  Call Extruder(568.39008)
  MoveL 7921 to (479.59, 455.55, 140) mm, rotated rx -180 ry 0 rz 160 deg; joints [0.602, 52.757, 6.65, -156.409, 61.55, 168.248]
  Set speed (16.6 mm/s)
  Call Extruder(574.71594)
  MoveL 7922 to (481.3, 454.8, 140) mm, rotated rx 180 ry 0 rz 160 deg; joints [0.5, 53.008, 6.147, -156.467, 61.298, 168.187]
  Set speed (16.6 mm/s)
  Call Extruder(580.66586)
  MoveL 7923 to (482.93, 454.17, 140) mm, rotated rx 180 ry 0 rz 160 deg; joints [0.414, 53.249, 5.663, -156.511, 61.059, 168.124]
  Set speed (16.6 mm/s)
  Call Extruder(586.68166)
  MoveL 7924 to (484.6, 453.58, 140) mm, rotated rx -180 ry 0 rz 160 deg; joints [0.335, 53.498, 5.165, -156.544, 60.813, 168.053]
  Set speed (16.6 mm/s)
  Call Extruder(592.98031)
  MoveL 7925 to (486.37, 453.02, 140) mm, rotated rx 180 ry 0 rz 160 deg; joints [0.261, 53.764, 4.634, -156.568, 60.554, 167.972]
  Call Extruder(599.08597)
  MoveL 7926 to (488.1, 452.56, 140) mm, rotated rx -180 ry 0 rz 160 deg; joints [0.198, 54.026, 4.11, -156.579, 60.301, 167.887]
  Set speed (16.6 mm/s)
  Call Extruder(605.30009)
  MoveL 7927 to (489.88, 452.15, 140) mm, rotated rx -180 ry 0 rz 160 deg; joints [0.144, 54.297, 3.568, -156.579, 60.042, 167.794]
  Set speed (16.6 mm/s)
  Call Extruder(611.23622)
  MoveL 7928 to (491.6, 451.81, 140) mm, rotated rx -180 ry 0 rz 160 deg; joints [0.1, 54.56, 3.044, -156.568, 59.792, 167.699]
  Set speed (16.6 mm/s)
  Call Extruder(617.09230)
  MoveL 7929 to (493.3, 451.55, 140) mm, rotated rx -180 ry 0 rz 160 deg; joints [0.065, 54.822, 2.521, -156.547, 59.545, 167.598]
  Call Extruder(623.59424)
  MoveL 7930 to (495.2, 451.32, 140) mm, rotated rx 180 ry 0 rz 160 deg; joints [0.036, 55.117, 1.933, -156.511, 59.27, 167.479]
  Set speed (16.6 mm/s)
  Call Extruder(629.59472)
  MoveL 7931 to (496.97, 451.18, 140) mm, rotated rx -180 ry 0 rz 160 deg; joints [0.018, 55.391, 1.386, -156.466, 59.016, 167.363]
  Set speed (16.6 mm/s)
  Call Extruder(635.88670)
  MoveL 7932 to (498.82, 451.1, 140) mm, rotated rx 180 ry 0 rz 160 deg; joints [0.008, 55.682, 0.807, -156.409, 58.75, 167.235]
  Call Extruder(641.91456)
  MoveL 7933 to (500.59, 451.09, 140) mm, rotated rx -180 ry 0 rz 160 deg; joints [0.006, 55.963, 0.248, -156.343, 58.495, 167.105]
  Set speed (16.6 mm/s)
  Call Extruder(648.10941)
  MoveL 7934 to (502.41, 451.15, 140) mm, rotated rx 180 ry 0 rz 160 deg; joints [0.013, 56.253, -0.329, -156.263, 58.234, 166.966]
  Set speed (16.6 mm/s)
  Call Extruder(654.14645)
  MoveL 7935 to (504.19, 451.27, 140) mm, rotated rx 180 ry 0 rz 160 deg; joints [0.028, 56.538, -0.895, -156.175, 57.98, 166.823]
  Set speed (16.6 mm/s)
  Call Extruder(660.34108)
  MoveL 7936 to (506, 451.46, 140) mm, rotated rx 180 ry 0 rz 160 deg; joints [0.052, 56.831, -1.477, -156.074, 57.721, 166.67]
  Set speed (16.6 mm/s)
  Call Extruder(666.29236)
  MoveL 7937 to (507.73, 451.71, 140) mm, rotated rx 180 ry 0 rz 160 deg; joints [0.083, 57.113, -2.037, -155.967, 57.474, 166.517]
  Call Extruder(672.33230)
  MoveL 7938 to (509.48, 452.02, 140) mm, rotated rx -180 ry 0 rz 160 deg; joints [0.122, 57.4, -2.606, -155.849, 57.226, 166.356]
  Set speed (16.6 mm/s)
  Call Extruder(678.01374)
  MoveL 7939 to (511.12, 452.37, 140) mm, rotated rx -180 ry 0 rz 160 deg; joints [0.165, 57.669, -3.141, -155.729, 56.994, 166.2]
  Set speed (16.6 mm/s)
  Call Extruder(684.72563)
  MoveL 7940 to (513.03, 452.85, 140) mm, rotated rx 180 ry 0 rz 160 deg; joints [0.224, 57.988, -3.772, -155.575, 56.724, 166.008]
  Set speed (16.6 mm/s)
  Call Extruder(690.75124)
  MoveL 7941 to (514.73, 453.36, 140) mm, rotated rx -180 ry 0 rz 160 deg; joints [0.286, 58.273, -4.336, -155.427, 56.484, 165.83]
  Set speed (16.6 mm/s)
  Call Extruder(697.05633)
  MoveL 7942 to (516.49, 453.95, 140) mm, rotated rx 180 ry 0 rz 160 deg; joints [0.358, 58.57, -4.925, -155.263, 56.237, 165.638]
  Set speed (16.6 mm/s)
  Call Extruder(702.95462)
  MoveL 7943 to (518.12, 454.57, 140) mm, rotated rx 180 ry 0 rz 160 deg; joints [0.432, 58.847, -5.472, -155.1, 56.01, 165.453]
  Set speed (16.6 mm/s)
  Call Extruder(709.29068)
  MoveL 7944 to (519.84, 455.29, 140) mm, rotated rx -180 ry 0 rz 160 deg; joints [0.519, 59.143, -6.057, -154.916, 55.77, 165.248]
  Set speed (16.6 mm/s)
  Call Extruder(715.36245)
  MoveL 7945 to (521.45, 456.04, 140) mm, rotated rx 180 ry 0 rz 160 deg; joints [0.609, 59.424, -6.612, -154.731, 55.545, 165.048]
  Set speed (16.6 mm/s)
  Call Extruder(721.45875)
  MoveL 7946 to (523.05, 456.86, 140) mm, rotated rx -180 ry 0 rz 160 deg; joints [0.706, 59.703, -7.163, -154.537, 55.324, 164.842]
  Set speed (16.6 mm/s)
  Call Extruder(727.63337)
  MoveL 7947 to (524.64, 457.75, 140) mm, rotated rx -180 ry 0 rz 160 deg; joints [0.81, 59.983, -7.716, -154.332, 55.106, 164.628]
  Set speed (16.6 mm/s)
  Call Extruder(733.66477)
  MoveL 7948 to (526.16, 458.67, 140) mm, rotated rx 180 ry 0 rz 160 deg; joints [0.919, 60.253, -8.249, -154.124, 54.898, 164.415]
  Set speed (16.6 mm/s)
  Call Extruder(739.87872)
  MoveL 7949 to (527.68, 459.68, 140) mm, rotated rx 180 ry 0 rz 160 deg; joints [1.037, 60.528, -8.791, -153.903, 54.69, 164.192]
  Set speed (16.6 mm/s)
  Call Extruder(745.90071)
  MoveL 7950 to (529.13, 460.7, 140) mm, rotated rx -180 ry 0 rz 160 deg; joints [1.157, 60.79, -9.307, -153.681, 54.495, 163.972]
  Call Extruder(751.89968)
  MoveL 7951 to (530.53, 461.78, 140) mm, rotated rx 180 ry 0 rz 160 deg; joints [1.282, 61.046, -9.812, -153.454, 54.307, 163.75]
  Set speed (16.6 mm/s)
  Call Extruder(758.13508)
  MoveL 7952 to (531.94, 462.95, 140) mm, rotated rx 180 ry 0 rz 160 deg; joints [1.418, 61.308, -10.327, -153.212, 54.119, 163.516]
  Set speed (16.6 mm/s)
  Call Extruder(764.34204)
  MoveL 7953 to (533.3, 464.17, 140) mm, rotated rx -180 ry 0 rz 160 deg; joints [1.559, 61.562, -10.829, -152.964, 53.939, 163.28]
  Set speed (16.6 mm/s)
  Call Extruder(770.41574)
  MoveL 7954 to (534.59, 465.41, 140) mm, rotated rx -180 ry 0 rz 160 deg; joints [1.701, 61.806, -11.308, -152.716, 53.771, 163.047]
  Set speed (16.6 mm/s)
  Call Extruder(773.76102)
  MoveL 7955 to (535.27, 466.12, 140) mm, rotated rx 180 ry 0 rz 160 deg; joints [1.782, 61.937, -11.566, -152.578, 53.681, 162.918]
  Set speed (16.6 mm/s)
  Call Extruder(776.78327)
  MoveL 7956 to (535.89, 466.76, 140) mm, rotated rx 180 ry 0 rz 160 deg; joints [1.856, 62.055, -11.797, -152.452, 53.602, 162.801]
  Set speed (16.6 mm/s)
  Call Extruder(780.49101)
  MoveL 7957 to (536.62, 467.57, 140) mm, rotated rx 180 ry 0 rz 160 deg; joints [1.948, 62.197, -12.076, -152.295, 53.509, 162.657]
  Set speed (16.6 mm/s)
  Call Extruder(783.96552)
  MoveL 7958 to (537.29, 468.35, 140) mm, rotated rx -180 ry 0 rz 160 deg; joints [2.037, 62.327, -12.332, -152.147, 53.424, 162.522]
  Set speed (16.6 mm/s)
  Call Extruder(786.90697)
  MoveL 7959 to (537.84, 469.01, 140) mm, rotated rx -180 ry 0 rz 160 deg; joints [2.112, 62.436, -12.546, -152.02, 53.354, 162.407]
  Set speed (16.6 mm/s)
  Call Extruder(790.76461)
  MoveL 7960 to (538.55, 469.9, 140) mm, rotated rx 180 ry 0 rz 160 deg; joints [2.213, 62.576, -12.821, -151.853, 53.265, 162.256]
  Call Extruder(794.10006)
  MoveL 7961 to (539.15, 470.68, 140) mm, rotated rx 180 ry 0 rz 160 deg; joints [2.302, 62.694, -13.053, -151.707, 53.192, 162.125]
  Set speed (16.6 mm/s)
  Call Extruder(797.30570)
  MoveL 7962 to (539.71, 471.44, 140) mm, rotated rx 180 ry 0 rz 160 deg; joints [2.388, 62.806, -13.273, -151.566, 53.123, 162]
  Set speed (16.6 mm/s)
  Call Extruder(800.87078)
  MoveL 7963 to (540.31, 472.3, 140) mm, rotated rx 180 ry 0 rz 160 deg; joints [2.486, 62.928, -13.513, -151.408, 53.05, 161.86]
  Set speed (16.6 mm/s)
  Call Extruder(804.35419)
  MoveL 7964 to (540.88, 473.15, 140) mm, rotated rx -180 ry 0 rz 160 deg; joints [2.582, 63.045, -13.742, -151.253, 52.982, 161.724]
  Set speed (16.6 mm/s)
  Call Extruder(807.31812)
  MoveL 7965 to (541.35, 473.88, 140) mm, rotated rx 180 ry 0 rz 160 deg; joints [2.665, 63.142, -13.932, -151.121, 52.926, 161.608]
  Call Extruder(811.18100)
  MoveL 7966 to (541.95, 474.85, 140) mm, rotated rx -180 ry 0 rz 160 deg; joints [2.774, 63.265, -14.174, -150.947, 52.857, 161.457]
  Set speed (16.6 mm/s)
  Call Extruder(816.88134)
  MoveL 7967 to (542.79, 476.3, 140) mm, rotated rx -180 ry 0 rz 160 deg; joints [2.938, 63.441, -14.519, -150.69, 52.762, 161.236]
  Set speed (16.6 mm/s)
  Call Extruder(821.30516)
  MoveL 7968 to (543.4, 477.44, 140) mm, rotated rx 180 ry 0 rz 160 deg; joints [3.067, 63.572, -14.776, -150.489, 52.694, 161.065]
  Set speed (16.6 mm/s)
  Call Extruder(824.85035)
  MoveL 7969 to (543.87, 478.38, 140) mm, rotated rx -180 ry 0 rz 160 deg; joints [3.172, 63.674, -14.976, -150.327, 52.643, 160.929]
  Set speed (16.6 mm/s)
  Call Extruder(829.78773)
  MoveL 7970 to (544.5, 479.69, 140) mm, rotated rx 180 ry 0 rz 160 deg; joints [3.32, 63.81, -15.243, -150.102, 52.578, 160.74]
  Set speed (16.6 mm/s)
  Call Extruder(831.57607)
  MoveL 7971 to (544.71, 480.17, 140) mm, rotated rx 180 ry 0 rz 160 deg; joints [3.374, 63.858, -15.336, -150.02, 52.556, 160.673]
  Set speed (16.6 mm/s)
  Call Extruder(838.17107)
  MoveL 7972 to (545.46, 481.95, 140) mm, rotated rx -180 ry 0 rz 160 deg; joints [3.575, 64.027, -15.667, -149.719, 52.483, 160.424]
  Set speed (16.6 mm/s)
  Call Extruder(843.12930)
  MoveL 7973 to (545.98, 483.32, 140) mm, rotated rx 180 ry 0 rz 160 deg; joints [3.728, 64.146, -15.901, -149.492, 52.436, 160.241]
  Set speed (16.6 mm/s)
  Call Extruder(845.31622)
  MoveL 7974 to (546.19, 483.92, 140) mm, rotated rx 180 ry 0 rz 160 deg; joints [3.797, 64.196, -15.999, -149.393, 52.417, 160.16]
  Set speed (16.6 mm/s)
  Call Extruder(851.93089)
  MoveL 7975 to (546.8, 485.77, 140) mm, rotated rx 180 ry 0 rz 160 deg; joints [4.005, 64.341, -16.283, -149.091, 52.369, 159.92]
  Set speed (16.6 mm/s)
  Call Extruder(855.40941)
  MoveL 7976 to (547.08, 486.76, 140) mm, rotated rx -180 ry 0 rz 160 deg; joints [4.115, 64.411, -16.421, -148.933, 52.349, 159.796]
  Set speed (16.6 mm/s)
  Call Extruder(858.85943)
  MoveL 7977 to (547.35, 487.73, 140) mm, rotated rx 180 ry 0 rz 160 deg; joints [4.225, 64.479, -16.553, -148.777, 52.332, 159.674]
  Set speed (16.6 mm/s)
  Call Extruder(865.59259)
  MoveL 7978 to (547.81, 489.66, 140) mm, rotated rx -180 ry 0 rz 160 deg; joints [4.442, 64.6, -16.791, -148.473, 52.308, 159.44]
  Set speed (16.6 mm/s)
  Call Extruder(872.38173)
  MoveL 7979 to (548.19, 491.62, 140) mm, rotated rx -180 ry 0 rz 160 deg; joints [4.664, 64.708, -17.002, -148.17, 52.299, 159.212]
  Set speed (16.6 mm/s)
  Call Extruder(879.18152)
  MoveL 7980 to (548.49, 493.6, 140) mm, rotated rx 180 ry 0 rz 160 deg; joints [4.887, 64.802, -17.187, -147.869, 52.302, 158.99]
  Set speed (16.6 mm/s)
  Call Extruder(886.08891)
  MoveL 7981 to (548.72, 495.62, 140) mm, rotated rx -180 ry 0 rz 160 deg; joints [5.115, 64.883, -17.344, -147.568, 52.319, 158.774]
  Call Extruder(892.76703)
  MoveL 7982 to (548.85, 497.58, 140) mm, rotated rx 180 ry 0 rz 160 deg; joints [5.338, 64.947, -17.47, -147.281, 52.348, 158.572]
  Set speed (16.6 mm/s)
  Call Extruder(899.57193)
  MoveL 7983 to (548.91, 499.59, 140) mm, rotated rx 180 ry 0 rz 160 deg; joints [5.565, 64.998, -17.568, -146.993, 52.391, 158.376]
  Set speed (16.6 mm/s)
  Call Extruder(906.22719)
  MoveL 7984 to (548.89, 501.55, 140) mm, rotated rx 180 ry 0 rz 160 deg; joints [5.789, 65.032, -17.636, -146.717, 52.446, 158.193]
  Set speed (16.6 mm/s)
  Call Extruder(913.15085)
  MoveL 7985 to (548.78, 503.58, 140) mm, rotated rx -180 ry 0 rz 160 deg; joints [6.022, 65.053, -17.677, -146.436, 52.516, 158.013]
  Set speed (16.6 mm/s)
  Call Extruder(919.94097)
  MoveL 7986 to (548.59, 505.57, 140) mm, rotated rx 180 ry 0 rz 160 deg; joints [6.251, 65.059, -17.688, -146.167, 52.598, 157.847]
  Set speed (16.6 mm/s)
  Call Extruder(926.85256)
  MoveL 7987 to (548.32, 507.59, 140) mm, rotated rx -180 ry 0 rz 160 deg; joints [6.483, 65.049, -17.669, -145.9, 52.694, 157.689]
  Set speed (16.6 mm/s)
  Call Extruder(933.53369)
  MoveL 7988 to (547.98, 509.53, 140) mm, rotated rx 180 ry 0 rz 160 deg; joints [6.708, 65.025, -17.622, -145.648, 52.798, 157.547]
  Set speed (16.6 mm/s)
  Call Extruder(940.45609)
  MoveL 7989 to (547.54, 511.52, 140) mm, rotated rx -180 ry 0 rz 160 deg; joints [6.94, 64.984, -17.542, -145.396, 52.919, 157.413]
  Set speed (16.6 mm/s)
  Call Extruder(947.08762)
  MoveL 7990 to (547.04, 513.41, 140) mm, rotated rx 180 ry 0 rz 160 deg; joints [7.162, 64.931, -17.438, -145.162, 53.046, 157.295]
  Set speed (16.6 mm/s)
  Call Extruder(949.76693)
  MoveL 7991 to (546.82, 514.16, 140) mm, rotated rx 180 ry 0 rz 160 deg; joints [7.251, 64.905, -17.387, -145.07, 53.101, 157.251]
  Set speed (16.6 mm/s)
  Call Extruder(953.95077)
  MoveL 7992 to (546.45, 515.34, 140) mm, rotated rx 180 ry 0 rz 160 deg; joints [7.39, 64.861, -17.301, -144.928, 53.189, 157.185]
  Set speed (16.6 mm/s)
  Call Extruder(960.63540)
  MoveL 7993 to (545.79, 517.19, 140) mm, rotated rx -180 ry 0 rz 160 deg; joints [7.61, 64.778, -17.139, -144.709, 53.34, 157.091]
  Set speed (16.6 mm/s)
  Call Extruder(964.14755)
  MoveL 7994 to (545.42, 518.15, 140) mm, rotated rx 180 ry 0 rz 160 deg; joints [7.725, 64.729, -17.043, -144.597, 53.423, 157.046]
  Set speed (16.6 mm/s)
  Call Extruder(967.44744)
  MoveL 7995 to (545.05, 519.05, 140) mm, rotated rx 180 ry 0 rz 160 deg; joints [7.833, 64.681, -16.948, -144.493, 53.503, 157.005]
  Set speed (16.6 mm/s)
  Call Extruder(974.29011)
  MoveL 7996 to (544.23, 520.89, 140) mm, rotated rx -180 ry 0 rz 160 deg; joints [8.056, 64.568, -16.727, -144.285, 53.678, 156.932]
  Set speed (16.6 mm/s)
  Call Extruder(977.80399)
  MoveL 7997 to (543.77, 521.82, 140) mm, rotated rx 180 ry 0 rz 160 deg; joints [8.169, 64.504, -16.603, -144.182, 53.772, 156.9]
  Set speed (16.6 mm/s)
  Call Extruder(981.05322)
  MoveL 7998 to (543.34, 522.68, 140) mm, rotated rx 180 ry 0 rz 160 deg; joints [8.273, 64.443, -16.482, -144.088, 53.861, 156.873]
  Set speed (16.6 mm/s)
  Call Extruder(984.45482)
  MoveL 7999 to (542.87, 523.56, 140) mm, rotated rx -180 ry 0 rz 160 deg; joints [8.382, 64.374, -16.349, -143.993, 53.956, 156.848]
  Set speed (16.6 mm/s)
  Call Extruder(987.85938)
  MoveL 8000 to (542.38, 524.43, 140) mm, rotated rx 180 ry 0 rz 160 deg; joints [8.49, 64.303, -16.209, -143.899, 54.054, 156.825]
  Set speed (16.6 mm/s)
  Call Extruder(992.09448)
  MoveL 8001 to (541.74, 525.5, 140) mm, rotated rx -180 ry 0 rz 160 deg; joints [8.623, 64.21, -16.027, -143.786, 54.178, 156.802]
  Set speed (16.6 mm/s)
  Call Extruder(997.75133)
  MoveL 8002 to (540.85, 526.91, 140) mm, rotated rx -180 ry 0 rz 160 deg; joints [8.799, 64.077, -15.767, -143.642, 54.35, 156.778]
  Set speed (16.6 mm/s)
  Call Extruder(1002.84044)
  MoveL 8003 to (540, 528.15, 140) mm, rotated rx 180 ry 0 rz 160 deg; joints [8.955, 63.951, -15.519, -143.516, 54.51, 156.764]
  Set speed (16.6 mm/s)
  Call Extruder(1008.25063)
  MoveL 8004 to (539.06, 529.43, 140) mm, rotated rx -180 ry 0 rz 160 deg; joints [9.119, 63.808, -15.239, -143.389, 54.684, 156.757]
  Set speed (16.6 mm/s)
  Call Extruder(1011.62355)
  MoveL 8005 to (538.46, 530.22, 140) mm, rotated rx 180 ry 0 rz 160 deg; joints [9.221, 63.716, -15.058, -143.313, 54.795, 156.756]
  Set speed (16.6 mm/s)
  Call Extruder(1015.04445)
  MoveL 8006 to (537.83, 531.01, 140) mm, rotated rx -180 ry 0 rz 160 deg; joints [9.322, 63.619, -14.868, -143.237, 54.91, 156.758]
  Set speed (16.6 mm/s)
  Call Extruder(1018.98481)
  MoveL 8007 to (537.08, 531.89, 140) mm, rotated rx -180 ry 0 rz 160 deg; joints [9.438, 63.504, -14.642, -143.154, 55.045, 156.764]
  Set speed (16.6 mm/s)
  Call Extruder(1025.23182)
  MoveL 8008 to (535.86, 533.27, 140) mm, rotated rx 180 ry 0 rz 160 deg; joints [9.619, 63.313, -14.269, -143.028, 55.262, 156.783]
  Set speed (16.6 mm/s)
  Call Extruder(1028.62384)
  MoveL 8009 to (535.17, 533.99, 140) mm, rotated rx 180 ry 0 rz 160 deg; joints [9.716, 63.206, -14.059, -142.963, 55.382, 156.796]
  Set speed (16.6 mm/s)
  Call Extruder(1031.99485)
  MoveL 8010 to (534.48, 534.7, 140) mm, rotated rx -180 ry 0 rz 160 deg; joints [9.811, 63.098, -13.846, -142.9, 55.503, 156.813]
  Call Extruder(1035.02733)
  MoveL 8011 to (533.84, 535.32, 140) mm, rotated rx -180 ry 0 rz 160 deg; joints [9.895, 62.997, -13.648, -142.846, 55.614, 156.831]
  Set speed (16.6 mm/s)
  Call Extruder(1038.77596)
  MoveL 8012 to (533.03, 536.08, 140) mm, rotated rx 180 ry 0 rz 160 deg; joints [9.999, 62.871, -13.4, -142.781, 55.752, 156.855]
  Call Extruder(1042.29481)
  MoveL 8013 to (532.26, 536.77, 140) mm, rotated rx 180 ry 0 rz 160 deg; joints [10.094, 62.749, -13.161, -142.723, 55.882, 156.881]
  Set speed (16.6 mm/s)
  Call Extruder(1045.62044)
  MoveL 8014 to (531.52, 537.4, 140) mm, rotated rx -180 ry 0 rz 160 deg; joints [10.183, 62.632, -12.931, -142.671, 56.007, 156.908]
  Set speed (16.6 mm/s)
  Call Extruder(1048.98991)
  MoveL 8015 to (530.75, 538.04, 140) mm, rotated rx 180 ry 0 rz 160 deg; joints [10.272, 62.511, -12.693, -142.62, 56.135, 156.939]
  Set speed (16.6 mm/s)
  Call Extruder(1051.88463)
  MoveL 8016 to (530.09, 538.57, 140) mm, rotated rx 180 ry 0 rz 160 deg; joints [10.347, 62.405, -12.485, -142.578, 56.245, 156.967]
  Call Extruder(1055.77726)
  MoveL 8017 to (529.17, 539.26, 140) mm, rotated rx -180 ry 0 rz 160 deg; joints [10.447, 62.26, -12.2, -142.525, 56.395, 157.008]
  Set speed (16.6 mm/s)
  Call Extruder(1059.25910)
  MoveL 8018 to (528.35, 539.86, 140) mm, rotated rx -180 ry 0 rz 160 deg; joints [10.534, 62.128, -11.941, -142.479, 56.531, 157.048]
  Set speed (16.6 mm/s)
  Call Extruder(1062.60815)
  MoveL 8019 to (527.54, 540.43, 140) mm, rotated rx 180 ry 0 rz 160 deg; joints [10.617, 61.999, -11.688, -142.438, 56.662, 157.088]
  Set speed (16.6 mm/s)
  Call Extruder(1066.01361)
  MoveL 8020 to (526.7, 540.98, 140) mm, rotated rx 180 ry 0 rz 160 deg; joints [10.7, 61.866, -11.426, -142.398, 56.796, 157.132]
  Set speed (16.6 mm/s)
  Call Extruder(1068.75461)
  MoveL 8021 to (526.02, 541.42, 140) mm, rotated rx 180 ry 0 rz 160 deg; joints [10.766, 61.757, -11.212, -142.368, 56.904, 157.169]
  Set speed (16.6 mm/s)
  Call Extruder(1073.72120)
  MoveL 8022 to (524.77, 542.18, 140) mm, rotated rx 180 ry 0 rz 160 deg; joints [10.882, 61.558, -10.82, -142.316, 57.102, 157.24]
  Set speed (16.6 mm/s)
  Call Extruder(1079.01856)
  MoveL 8023 to (523.42, 542.95, 140) mm, rotated rx 180 ry 0 rz 160 deg; joints [11.002, 61.341, -10.392, -142.267, 57.315, 157.322]
  Set speed (16.6 mm/s)
  Call Extruder(1085.08509)
  MoveL 8024 to (521.84, 543.77, 140) mm, rotated rx 180 ry 0 rz 160 deg; joints [11.135, 61.088, -9.894, -142.218, 57.56, 157.421]
  Set speed (16.6 mm/s)
  Call Extruder(1089.75809)
  MoveL 8025 to (520.6, 544.37, 140) mm, rotated rx 180 ry 0 rz 160 deg; joints [11.233, 60.889, -9.502, -142.185, 57.75, 157.504]
  Set speed (16.6 mm/s)
  Call Extruder(1096.60033)
  MoveL 8026 to (518.75, 545.18, 140) mm, rotated rx -180 ry 0 rz 160 deg; joints [11.372, 60.593, -8.919, -142.145, 58.03, 157.632]
  Set speed (16.6 mm/s)
  Call Extruder(1103.38214)
  MoveL 8027 to (516.89, 545.9, 140) mm, rotated rx -180 ry 0 rz 160 deg; joints [11.502, 60.294, -8.33, -142.114, 58.308, 157.767]
  Set speed (16.6 mm/s)
  Call Extruder(1110.16826)
  MoveL 8028 to (515.01, 546.55, 140) mm, rotated rx -180 ry 0 rz 160 deg; joints [11.624, 59.99, -7.731, -142.092, 58.588, 157.91]
  Set speed (16.6 mm/s)
  Call Extruder(1116.92882)
  MoveL 8029 to (513.1, 547.13, 140) mm, rotated rx 180 ry 0 rz 160 deg; joints [11.739, 59.684, -7.126, -142.079, 58.866, 158.06]
  Set speed (16.6 mm/s)
  Call Extruder(1118.77020)
  MoveL 8030 to (512.58, 547.27, 140) mm, rotated rx -180 ry 0 rz 160 deg; joints [11.769, 59.6, -6.96, -142.077, 58.942, 158.102]
  Set speed (16.6 mm/s)
  Call Extruder(1123.83770)
  MoveL 8031 to (511.13, 547.63, 140) mm, rotated rx -180 ry 0 rz 160 deg; joints [11.848, 59.367, -6.501, -142.075, 59.15, 158.221]
  Set speed (16.6 mm/s)
  Call Extruder(1130.70374)
  MoveL 8032 to (509.16, 548.05, 140) mm, rotated rx -180 ry 0 rz 160 deg; joints [11.948, 59.049, -5.872, -142.081, 59.432, 158.387]
  Set speed (16.6 mm/s)
  Call Extruder(1137.39674)
  MoveL 8033 to (507.22, 548.38, 140) mm, rotated rx 180 ry 0 rz 160 deg; joints [12.036, 58.736, -5.253, -142.096, 59.706, 158.557]
  Call Extruder(1144.16481)
  MoveL 8034 to (505.24, 548.63, 140) mm, rotated rx -180 ry 0 rz 160 deg; joints [12.118, 58.418, -4.623, -142.119, 59.981, 158.734]
  Set speed (16.6 mm/s)
  Call Extruder(1151.12946)
  MoveL 8035 to (503.2, 548.81, 140) mm, rotated rx -180 ry 0 rz 160 deg; joints [12.192, 58.089, -3.971, -142.153, 60.263, 158.923]
  Call Extruder(1157.97300)
  MoveL 8036 to (501.19, 548.9, 140) mm, rotated rx -180 ry 0 rz 160 deg; joints [12.256, 57.764, -3.329, -142.195, 60.537, 159.113]
  Set speed (16.6 mm/s)
  Call Extruder(1164.59319)
  MoveL 8037 to (499.24, 548.91, 140) mm, rotated rx -180 ry 0 rz 160 deg; joints [12.309, 57.45, -2.705, -142.245, 60.8, 159.303]
  Set speed (10.0 mm/s)
  MoveL 8038 to (499.24, 548.91, 144) mm, rotated rx -180 ry 0 rz 160 deg; joints [12.309, 56.866, -2.538, -142.101, 60.471, 159.01]
  Set speed (120.0 mm/s)
  MoveL 8039 to (499.24, 547.28, 144) mm, rotated rx 180 ry 0 rz 160 deg; joints [12.11, 56.809, -2.426, -142.334, 60.444, 159.154]
  Set speed (16.7 mm/s)
  Call Extruder(1171.18719)
  MoveL 8040 to (497.29, 547.21, 144) mm, rotated rx 180 ry 0 rz 160 deg; joints [12.152, 56.492, -1.801, -142.394, 60.702, 159.347]
  Call Extruder(1177.73544)
  MoveL 8041 to (495.35, 547.05, 144) mm, rotated rx -180 ry 0 rz 160 deg; joints [12.185, 56.178, -1.181, -142.463, 60.956, 159.544]
  Set speed (16.7 mm/s)
  Call Extruder(1184.19711)
  MoveL 8042 to (493.45, 546.83, 144) mm, rotated rx 180 ry 0 rz 160 deg; joints [12.208, 55.868, -0.571, -142.54, 61.203, 159.741]
  Set speed (16.7 mm/s)
  Call Extruder(1190.67402)
  MoveL 8043 to (491.55, 546.52, 144) mm, rotated rx 180 ry 0 rz 160 deg; joints [12.221, 55.56, 0.039, -142.626, 61.447, 159.943]
  Call Extruder(1197.03784)
  MoveL 8044 to (489.7, 546.15, 144) mm, rotated rx -180 ry 0 rz 160 deg; joints [12.224, 55.258, 0.635, -142.719, 61.682, 160.144]
  Set speed (16.7 mm/s)
  Call Extruder(1200.54963)
  MoveL 8045 to (488.69, 545.91, 144) mm, rotated rx -180 ry 0 rz 160 deg; joints [12.221, 55.093, 0.962, -142.775, 61.809, 160.257]
  Call Extruder(1203.76062)
  MoveL 8046 to (487.77, 545.67, 144) mm, rotated rx -180 ry 0 rz 160 deg; joints [12.217, 54.942, 1.259, -142.827, 61.925, 160.36]
  Set speed (16.7 mm/s)
  Call Extruder(1210.22712)
  MoveL 8047 to (485.93, 545.14, 144) mm, rotated rx -180 ry 0 rz 160 deg; joints [12.2, 54.641, 1.856, -142.939, 62.154, 160.569]
  Call Extruder(1216.71711)
  MoveL 8048 to (484.1, 544.53, 144) mm, rotated rx -180 ry 0 rz 160 deg; joints [12.173, 54.341, 2.448, -143.061, 62.379, 160.782]
  Set speed (16.7 mm/s)
  Call Extruder(1220.14720)
  MoveL 8049 to (483.15, 544.18, 144) mm, rotated rx 180 ry 0 rz 160 deg; joints [12.154, 54.185, 2.758, -143.129, 62.496, 160.895]
  Set speed (16.7 mm/s)
  Call Extruder(1224.84220)
  MoveL 8050 to (481.86, 543.67, 144) mm, rotated rx -180 ry 0 rz 160 deg; joints [12.125, 53.972, 3.178, -143.225, 62.653, 161.05]
  Set speed (16.7 mm/s)
  Call Extruder(1230.35260)
  MoveL 8051 to (480.37, 543.02, 144) mm, rotated rx 180 ry 0 rz 160 deg; joints [12.083, 53.726, 3.667, -143.344, 62.833, 161.233]
  Set speed (16.7 mm/s)
  Call Extruder(1233.09228)
  MoveL 8052 to (479.63, 542.67, 144) mm, rotated rx 180 ry 0 rz 160 deg; joints [12.059, 53.604, 3.908, -143.406, 62.921, 161.325]
  Set speed (16.7 mm/s)
  Call Extruder(1236.38565)
  MoveL 8053 to (478.75, 542.24, 144) mm, rotated rx 180 ry 0 rz 160 deg; joints [12.028, 53.459, 4.195, -143.483, 63.026, 161.435]
  Set speed (16.7 mm/s)
  Call Extruder(1239.73406)
  MoveL 8054 to (477.87, 541.79, 144) mm, rotated rx 180 ry 0 rz 160 deg; joints [11.994, 53.313, 4.485, -143.562, 63.131, 161.548]
  Call Extruder(1242.83206)
  MoveL 8055 to (477.06, 541.35, 144) mm, rotated rx 180 ry 0 rz 160 deg; joints [11.959, 53.179, 4.751, -143.638, 63.226, 161.652]
  Set speed (16.7 mm/s)
  Call Extruder(1246.17560)
  MoveL 8056 to (476.2, 540.86, 144) mm, rotated rx 180 ry 0 rz 160 deg; joints [11.92, 53.036, 5.035, -143.723, 63.327, 161.764]
  Call Extruder(1249.42346)
  MoveL 8057 to (475.38, 540.37, 144) mm, rotated rx -180 ry 0 rz 160 deg; joints [11.879, 52.898, 5.308, -143.806, 63.424, 161.873]
  Set speed (16.7 mm/s)
  Call Extruder(1254.36238)
  MoveL 8058 to (474.14, 539.59, 144) mm, rotated rx 180 ry 0 rz 160 deg; joints [11.811, 52.691, 5.719, -143.938, 63.567, 162.04]
  Call Extruder(1259.18569)
  MoveL 8059 to (472.95, 538.78, 144) mm, rotated rx 180 ry 0 rz 160 deg; joints [11.739, 52.493, 6.114, -144.072, 63.704, 162.202]
  Set speed (16.7 mm/s)
  Call Extruder(1262.45339)
  MoveL 8060 to (472.16, 538.22, 144) mm, rotated rx -180 ry 0 rz 160 deg; joints [11.687, 52.36, 6.377, -144.165, 63.794, 162.312]
  Set speed (16.7 mm/s)
  Call Extruder(1265.82623)
  MoveL 8061 to (471.36, 537.62, 144) mm, rotated rx -180 ry 0 rz 160 deg; joints [11.631, 52.225, 6.646, -144.263, 63.885, 162.426]
  Set speed (16.7 mm/s)
  Call Extruder(1268.90857)
  MoveL 8062 to (470.64, 537.06, 144) mm, rotated rx 180 ry 0 rz 160 deg; joints [11.577, 52.103, 6.888, -144.354, 63.967, 162.529]
  Set speed (16.7 mm/s)
  Call Extruder(1272.86798)
  MoveL 8063 to (469.73, 536.32, 144) mm, rotated rx 180 ry 0 rz 160 deg; joints [11.504, 51.949, 7.195, -144.475, 64.069, 162.661]
  Set speed (16.7 mm/s)
  Call Extruder(1275.51804)
  MoveL 8064 to (469.13, 535.81, 144) mm, rotated rx -180 ry 0 rz 160 deg; joints [11.453, 51.847, 7.397, -144.557, 64.136, 162.75]
  Set speed (16.7 mm/s)
  Call Extruder(1278.84572)
  MoveL 8065 to (468.39, 535.16, 144) mm, rotated rx 180 ry 0 rz 160 deg; joints [11.387, 51.721, 7.648, -144.662, 64.218, 162.861]
  Call Extruder(1281.96684)
  MoveL 8066 to (467.7, 534.54, 144) mm, rotated rx 180 ry 0 rz 160 deg; joints [11.322, 51.605, 7.88, -144.763, 64.293, 162.965]
  Set speed (16.7 mm/s)
  Call Extruder(1284.91732)
  MoveL 8067 to (467.07, 533.93, 144) mm, rotated rx -180 ry 0 rz 160 deg; joints [11.259, 51.496, 8.096, -144.86, 64.363, 163.062]
  Call Extruder(1288.53930)
  MoveL 8068 to (466.31, 533.17, 144) mm, rotated rx 180 ry 0 rz 160 deg; joints [11.179, 51.365, 8.357, -144.981, 64.445, 163.182]
  Set speed (16.7 mm/s)
  Call Extruder(1291.89779)
  MoveL 8069 to (465.62, 532.46, 144) mm, rotated rx -180 ry 0 rz 160 deg; joints [11.102, 51.246, 8.594, -145.095, 64.52, 163.292]
  Set speed (16.7 mm/s)
  Call Extruder(1295.01891)
  MoveL 8070 to (464.99, 531.78, 144) mm, rotated rx -180 ry 0 rz 160 deg; joints [11.028, 51.137, 8.811, -145.203, 64.587, 163.394]
  Set speed (16.7 mm/s)
  Call Extruder(1298.28206)
  MoveL 8071 to (464.34, 531.06, 144) mm, rotated rx 180 ry 0 rz 160 deg; joints [10.948, 51.025, 9.033, -145.317, 64.656, 163.5]
  Set speed (16.7 mm/s)
  Call Extruder(1301.61667)
  MoveL 8072 to (463.7, 530.3, 144) mm, rotated rx 180 ry 0 rz 160 deg; joints [10.864, 50.914, 9.256, -145.436, 64.724, 163.608]
  Set speed (16.7 mm/s)
  Call Extruder(1304.77781)
  MoveL 8073 to (463.11, 529.58, 144) mm, rotated rx -180 ry 0 rz 160 deg; joints [10.782, 50.809, 9.464, -145.551, 64.786, 163.71]
  Set speed (16.7 mm/s)
  Call Extruder(1308.09321)
  MoveL 8074 to (462.51, 528.8, 144) mm, rotated rx -180 ry 0 rz 160 deg; joints [10.694, 50.703, 9.676, -145.673, 64.848, 163.816]
  Call Extruder(1311.34058)
  MoveL 8075 to (461.92, 528.04, 144) mm, rotated rx 180 ry 0 rz 160 deg; joints [10.605, 50.6, 9.881, -145.794, 64.908, 163.92]
  Set speed (16.7 mm/s)
  Call Extruder(1314.63787)
  MoveL 8076 to (461.35, 527.24, 144) mm, rotated rx -180 ry 0 rz 160 deg; joints [10.512, 50.499, 10.083, -145.919, 64.966, 164.024]
  Set speed (16.7 mm/s)
  Call Extruder(1317.91073)
  MoveL 8077 to (460.8, 526.44, 144) mm, rotated rx 180 ry 0 rz 160 deg; joints [10.418, 50.4, 10.28, -146.044, 65.021, 164.127]
  Call Extruder(1321.12803)
  MoveL 8078 to (460.28, 525.65, 144) mm, rotated rx -180 ry 0 rz 160 deg; joints [10.324, 50.306, 10.469, -146.169, 65.074, 164.227]
  Set speed (16.7 mm/s)
  Call Extruder(1324.43377)
  MoveL 8079 to (459.75, 524.82, 144) mm, rotated rx 180 ry 0 rz 160 deg; joints [10.224, 50.211, 10.657, -146.299, 65.125, 164.329]
  Set speed (16.7 mm/s)
  Call Extruder(1327.65036)
  MoveL 8080 to (459.26, 524, 144) mm, rotated rx 180 ry 0 rz 160 deg; joints [10.125, 50.122, 10.837, -146.427, 65.173, 164.428]
  Set speed (16.7 mm/s)
  Call Extruder(1330.95898)
  MoveL 8081 to (458.77, 523.15, 144) mm, rotated rx 180 ry 0 rz 160 deg; joints [10.021, 50.032, 11.015, -146.56, 65.22, 164.528]
  Set speed (16.7 mm/s)
  Call Extruder(1334.18242)
  MoveL 8082 to (458.31, 522.31, 144) mm, rotated rx -180 ry 0 rz 160 deg; joints [9.918, 49.947, 11.185, -146.691, 65.263, 164.626]
  Call Extruder(1337.66472)
  MoveL 8083 to (457.84, 521.4, 144) mm, rotated rx 180 ry 0 rz 160 deg; joints [9.804, 49.858, 11.362, -146.834, 65.307, 164.729]
  Call Extruder(1340.68804)
  MoveL 8084 to (457.44, 520.59, 144) mm, rotated rx 180 ry 0 rz 160 deg; joints [9.704, 49.784, 11.511, -146.96, 65.343, 164.819]
  Set speed (16.7 mm/s)
  Call Extruder(1344.07923)
  MoveL 8085 to (457.01, 519.68, 144) mm, rotated rx 180 ry 0 rz 160 deg; joints [9.589, 49.703, 11.673, -147.102, 65.381, 164.918]
  Set speed (16.7 mm/s)
  Call Extruder(1347.17208)
  MoveL 8086 to (456.64, 518.85, 144) mm, rotated rx 180 ry 0 rz 160 deg; joints [9.483, 49.631, 11.816, -147.232, 65.414, 165.008]
  Set speed (16.7 mm/s)
  Call Extruder(1353.89946)
  MoveL 8087 to (455.88, 517, 144) mm, rotated rx 180 ry 0 rz 160 deg; joints [9.247, 49.484, 12.111, -147.52, 65.477, 165.199]
  Set speed (16.7 mm/s)
  Call Extruder(1360.28373)
  MoveL 8088 to (455.23, 515.22, 144) mm, rotated rx 180 ry 0 rz 160 deg; joints [9.015, 49.355, 12.369, -147.797, 65.527, 165.377]
  Set speed (16.7 mm/s)
  Call Extruder(1366.77671)
  MoveL 8089 to (454.65, 513.39, 144) mm, rotated rx 180 ry 0 rz 160 deg; joints [8.774, 49.235, 12.61, -148.083, 65.568, 165.554]
  Set speed (16.7 mm/s)
  Call Extruder(1370.18077)
  MoveL 8090 to (454.38, 512.42, 144) mm, rotated rx 180 ry 0 rz 160 deg; joints [8.645, 49.177, 12.726, -148.233, 65.586, 165.644]
  Set speed (16.7 mm/s)
  Call Extruder(1373.44164)
  MoveL 8091 to (454.13, 511.48, 144) mm, rotated rx 180 ry 0 rz 160 deg; joints [8.521, 49.123, 12.833, -148.379, 65.601, 165.73]
  Set speed (16.7 mm/s)
  Call Extruder(1379.87855)
  MoveL 8092 to (453.71, 509.62, 144) mm, rotated rx -180 ry 0 rz 160 deg; joints [8.271, 49.026, 13.027, -148.667, 65.622, 165.895]
  Set speed (16.7 mm/s)
  Call Extruder(1386.53127)
  MoveL 8093 to (453.34, 507.69, 144) mm, rotated rx 180 ry 0 rz 160 deg; joints [8.008, 48.938, 13.203, -148.968, 65.634, 166.061]
  Call Extruder(1392.79064)
  MoveL 8094 to (453.08, 505.85, 144) mm, rotated rx 180 ry 0 rz 160 deg; joints [7.756, 48.867, 13.346, -149.253, 65.635, 166.212]
  Set speed (16.7 mm/s)
  Call Extruder(1399.57375)
  MoveL 8095 to (452.87, 503.85, 144) mm, rotated rx 180 ry 0 rz 160 deg; joints [7.48, 48.802, 13.477, -149.562, 65.626, 166.37]
  Set speed (16.7 mm/s)
  Call Extruder(1406.06382)
  MoveL 8096 to (452.76, 501.93, 144) mm, rotated rx 180 ry 0 rz 160 deg; joints [7.213, 48.752, 13.577, -149.859, 65.607, 166.515]
  Set speed (16.7 mm/s)
  Call Extruder(1412.52517)
  MoveL 8097 to (452.72, 500.01, 144) mm, rotated rx -180 ry 0 rz 160 deg; joints [6.945, 48.714, 13.652, -150.154, 65.577, 166.654]
  Set speed (16.7 mm/s)
  Call Extruder(1418.49455)
  MoveL 8098 to (452.75, 498.25, 144) mm, rotated rx 180 ry 0 rz 160 deg; joints [6.696, 48.689, 13.703, -150.426, 65.542, 166.778]
  Set speed (16.7 mm/s)
  Call Extruder(1424.19299)
  MoveL 8099 to (452.84, 496.56, 144) mm, rotated rx -180 ry 0 rz 160 deg; joints [6.458, 48.675, 13.731, -150.684, 65.5, 166.891]
  Set speed (16.7 mm/s)
  Call Extruder(1430.13443)
  MoveL 8100 to (453, 494.8, 144) mm, rotated rx 180 ry 0 rz 160 deg; joints [6.208, 48.67, 13.74, -150.952, 65.448, 167.005]
  Call Extruder(1436.00568)
  MoveL 8101 to (453.23, 493.08, 144) mm, rotated rx 180 ry 0 rz 160 deg; joints [5.962, 48.676, 13.729, -151.215, 65.388, 167.112]
  Call Extruder(1441.97681)
  MoveL 8102 to (453.52, 491.33, 144) mm, rotated rx -180 ry 0 rz 160 deg; joints [5.712, 48.691, 13.698, -151.48, 65.319, 167.215]
  Set speed (16.7 mm/s)
  Call Extruder(1447.75941)
  MoveL 8103 to (453.86, 489.65, 144) mm, rotated rx -180 ry 0 rz 160 deg; joints [5.471, 48.716, 13.649, -151.734, 65.244, 167.311]
  Call Extruder(1453.62597)
  MoveL 8104 to (454.27, 487.96, 144) mm, rotated rx 180 ry 0 rz 160 deg; joints [5.227, 48.751, 13.578, -151.987, 65.159, 167.402]
  Set speed (16.7 mm/s)
  Call Extruder(1459.39877)
  MoveL 8105 to (454.74, 486.32, 144) mm, rotated rx -180 ry 0 rz 160 deg; joints [4.99, 48.795, 13.49, -152.234, 65.068, 167.487]
  Call Extruder(1465.30030)
  MoveL 8106 to (455.28, 484.65, 144) mm, rotated rx 180 ry 0 rz 160 deg; joints [4.749, 48.85, 13.381, -152.481, 64.968, 167.568]
  Set speed (16.7 mm/s)
  Call Extruder(1471.24681)
  MoveL 8107 to (455.88, 483, 144) mm, rotated rx 180 ry 0 rz 160 deg; joints [4.509, 48.915, 13.25, -152.725, 64.858, 167.645]
  Set speed (16.7 mm/s)
  Call Extruder(1476.18883)
  MoveL 8108 to (456.43, 481.64, 144) mm, rotated rx -180 ry 0 rz 160 deg; joints [4.313, 48.976, 13.127, -152.925, 64.762, 167.704]
  Set speed (16.7 mm/s)
  Call Extruder(1482.90047)
  MoveL 8109 to (457.24, 479.82, 144) mm, rotated rx -180 ry 0 rz 160 deg; joints [4.049, 49.07, 12.939, -153.189, 64.622, 167.778]
  Set speed (16.7 mm/s)
  Call Extruder(1488.70804)
  MoveL 8110 to (458, 478.28, 144) mm, rotated rx 180 ry 0 rz 160 deg; joints [3.826, 49.162, 12.756, -153.411, 64.493, 167.837]
  Set speed (16.7 mm/s)
  Call Extruder(1494.73356)
  MoveL 8111 to (458.85, 476.71, 144) mm, rotated rx 180 ry 0 rz 160 deg; joints [3.598, 49.266, 12.547, -153.636, 64.351, 167.892]
  Call Extruder(1500.69829)
  MoveL 8112 to (459.75, 475.19, 144) mm, rotated rx 180 ry 0 rz 160 deg; joints [3.378, 49.379, 12.321, -153.851, 64.204, 167.94]
  Set speed (16.7 mm/s)
  Call Extruder(1506.48572)
  MoveL 8113 to (460.68, 473.74, 144) mm, rotated rx 180 ry 0 rz 160 deg; joints [3.169, 49.497, 12.085, -154.053, 64.054, 167.981]
  Set speed (16.7 mm/s)
  Call Extruder(1512.35919)
  MoveL 8114 to (461.67, 472.31, 144) mm, rotated rx -180 ry 0 rz 160 deg; joints [2.962, 49.626, 11.827, -154.25, 63.895, 168.018]
  Set speed (16.7 mm/s)
  Call Extruder(1518.30667)
  MoveL 8115 to (462.73, 470.9, 144) mm, rotated rx 180 ry 0 rz 160 deg; joints [2.759, 49.765, 11.549, -154.442, 63.728, 168.048]
  Call Extruder(1524.02029)
  MoveL 8116 to (463.8, 469.59, 144) mm, rotated rx -180 ry 0 rz 160 deg; joints [2.57, 49.907, 11.264, -154.618, 63.56, 168.072]
  Set speed (16.7 mm/s)
  Call Extruder(1529.82101)
  MoveL 8117 to (464.93, 468.29, 144) mm, rotated rx 180 ry 0 rz 160 deg; joints [2.384, 50.06, 10.96, -154.789, 63.384, 168.09]
  Set speed (16.7 mm/s)
  Call Extruder(1535.93421)
  MoveL 8118 to (466.17, 466.97, 144) mm, rotated rx -180 ry 0 rz 160 deg; joints [2.195, 50.229, 10.623, -154.96, 63.193, 168.103]
  Set speed (16.7 mm/s)
  Call Extruder(1541.70205)
  MoveL 8119 to (467.39, 465.76, 144) mm, rotated rx 180 ry 0 rz 160 deg; joints [2.024, 50.396, 10.288, -155.113, 63.006, 168.109]
  Call Extruder(1547.41065)
  MoveL 8120 to (468.63, 464.62, 144) mm, rotated rx -180 ry 0 rz 160 deg; joints [1.861, 50.569, 9.943, -155.254, 62.816, 168.109]
  Set speed (16.7 mm/s)
  Call Extruder(1553.53237)
  MoveL 8121 to (470.01, 463.44, 144) mm, rotated rx -180 ry 0 rz 160 deg; joints [1.694, 50.763, 9.557, -155.397, 62.607, 168.103]
  Call Extruder(1559.32388)
  MoveL 8122 to (471.36, 462.38, 144) mm, rotated rx 180 ry 0 rz 160 deg; joints [1.543, 50.953, 9.178, -155.522, 62.404, 168.091]
  Set speed (16.7 mm/s)
  Call Extruder(1565.18702)
  MoveL 8123 to (472.76, 461.35, 144) mm, rotated rx 180 ry 0 rz 160 deg; joints [1.399, 51.153, 8.78, -155.639, 62.194, 168.073]
  Call Extruder(1570.97827)
  MoveL 8124 to (474.19, 460.39, 144) mm, rotated rx -180 ry 0 rz 160 deg; joints [1.264, 51.357, 8.373, -155.744, 61.982, 168.049]
  Call Extruder(0.00000)
  Set speed (16.7 mm/s)
  Call Extruder(6.02801)
  MoveL 8125 to (475.7, 459.44, 144) mm, rotated rx 180 ry 0 rz 160 deg; joints [1.132, 51.576, 7.937, -155.843, 61.756, 168.017]
  Set speed (16.7 mm/s)
  Call Extruder(11.90523)
  MoveL 8126 to (477.21, 458.57, 144) mm, rotated rx 180 ry 0 rz 160 deg; joints [1.011, 51.796, 7.5, -155.929, 61.532, 167.979]
  Call Extruder(17.73477)
  MoveL 8127 to (478.74, 457.77, 144) mm, rotated rx -180 ry 0 rz 160 deg; joints [0.9, 52.02, 7.054, -156.004, 61.307, 167.936]
  Set speed (16.7 mm/s)
  Call Extruder(23.48475)
  MoveL 8128 to (480.28, 457.03, 144) mm, rotated rx -180 ry 0 rz 160 deg; joints [0.798, 52.246, 6.604, -156.067, 61.081, 167.887]
  Set speed (16.7 mm/s)
  Call Extruder(29.25314)
  MoveL 8129 to (481.84, 456.34, 144) mm, rotated rx 180 ry 0 rz 160 deg; joints [0.704, 52.478, 6.142, -156.121, 60.851, 167.832]
  Set speed (16.7 mm/s)
  Call Extruder(35.22799)
  MoveL 8130 to (483.49, 455.69, 144) mm, rotated rx 180 ry 0 rz 160 deg; joints [0.616, 52.724, 5.653, -156.165, 60.611, 167.768]
  Set speed (16.7 mm/s)
  Call Extruder(41.26768)
  MoveL 8131 to (485.18, 455.1, 144) mm, rotated rx 180 ry 0 rz 160 deg; joints [0.535, 52.978, 5.149, -156.198, 60.365, 167.696]
  Set speed (16.7 mm/s)
  Call Extruder(46.96001)
  MoveL 8132 to (486.79, 454.6, 144) mm, rotated rx -180 ry 0 rz 160 deg; joints [0.467, 53.222, 4.666, -156.219, 60.131, 167.622]
  Set speed (16.7 mm/s)
  Call Extruder(53.02574)
  MoveL 8133 to (488.53, 454.13, 144) mm, rotated rx 180 ry 0 rz 160 deg; joints [0.404, 53.486, 4.142, -156.23, 59.88, 167.537]
  Call Extruder(58.79823)
  MoveL 8134 to (490.19, 453.74, 144) mm, rotated rx -180 ry 0 rz 160 deg; joints [0.352, 53.742, 3.636, -156.23, 59.639, 167.45]
  Set speed (16.7 mm/s)
  Call Extruder(64.66585)
  MoveL 8135 to (491.9, 453.42, 144) mm, rotated rx -180 ry 0 rz 160 deg; joints [0.308, 54.005, 3.114, -156.219, 59.393, 167.354]
  Set speed (16.7 mm/s)
  Call Extruder(70.56866)
  MoveL 8136 to (493.63, 453.15, 144) mm, rotated rx -180 ry 0 rz 160 deg; joints [0.272, 54.273, 2.583, -156.196, 59.144, 167.251]
  Call Extruder(76.49937)
  MoveL 8137 to (495.38, 452.95, 144) mm, rotated rx -180 ry 0 rz 160 deg; joints [0.245, 54.546, 2.043, -156.162, 58.894, 167.142]
  Set speed (16.7 mm/s)
  Call Extruder(82.21045)
  MoveL 8138 to (497.07, 452.81, 144) mm, rotated rx -180 ry 0 rz 160 deg; joints [0.227, 54.811, 1.518, -156.119, 58.652, 167.03]
  Set speed (16.7 mm/s)
  Call Extruder(88.24453)
  MoveL 8139 to (498.86, 452.73, 144) mm, rotated rx -180 ry 0 rz 160 deg; joints [0.216, 55.094, 0.959, -156.063, 58.397, 166.905]
  Set speed (16.7 mm/s)
  Call Extruder(94.03135)
  MoveL 8140 to (500.57, 452.72, 144) mm, rotated rx 180 ry 0 rz 160 deg; joints [0.214, 55.367, 0.419, -155.999, 58.153, 166.779]
  Call Extruder(99.96574)
  MoveL 8141 to (502.33, 452.77, 144) mm, rotated rx 180 ry 0 rz 160 deg; joints [0.22, 55.65, -0.139, -155.922, 57.903, 166.643]
  Call Extruder(105.76897)
  MoveL 8142 to (504.05, 452.89, 144) mm, rotated rx 180 ry 0 rz 160 deg; joints [0.233, 55.927, -0.686, -155.837, 57.66, 166.504]
  Set speed (16.7 mm/s)
  Call Extruder(111.71053)
  MoveL 8143 to (505.8, 453.07, 144) mm, rotated rx -180 ry 0 rz 160 deg; joints [0.256, 56.212, -1.248, -155.739, 57.412, 166.356]
  Set speed (16.7 mm/s)
  Call Extruder(117.41040)
  MoveL 8144 to (507.48, 453.31, 144) mm, rotated rx 180 ry 0 rz 160 deg; joints [0.285, 56.485, -1.788, -155.635, 57.177, 166.207]
  Call Extruder(123.36081)
  MoveL 8145 to (509.21, 453.62, 144) mm, rotated rx 180 ry 0 rz 160 deg; joints [0.322, 56.772, -2.352, -155.517, 56.932, 166.047]
  Call Extruder(129.09442)
  MoveL 8146 to (510.87, 453.98, 144) mm, rotated rx -180 ry 0 rz 160 deg; joints [0.366, 57.047, -2.895, -155.393, 56.7, 165.886]
  Set speed (16.7 mm/s)
  Call Extruder(135.01581)
  MoveL 8147 to (512.58, 454.42, 144) mm, rotated rx -180 ry 0 rz 160 deg; joints [0.419, 57.332, -3.455, -155.256, 56.462, 165.714]
  Call Extruder(140.98986)
  MoveL 8148 to (514.27, 454.92, 144) mm, rotated rx -180 ry 0 rz 160 deg; joints [0.479, 57.618, -4.018, -155.108, 56.226, 165.536]
  Set speed (16.7 mm/s)
  Call Extruder(146.92211)
  MoveL 8149 to (515.94, 455.49, 144) mm, rotated rx 180 ry 0 rz 160 deg; joints [0.547, 57.901, -4.575, -154.952, 55.995, 165.353]
  Set speed (16.7 mm/s)
  Call Extruder(152.71074)
  MoveL 8150 to (517.54, 456.09, 144) mm, rotated rx 180 ry 0 rz 160 deg; joints [0.62, 58.175, -5.115, -154.79, 55.773, 165.169]
  Call Extruder(158.67352)
  MoveL 8151 to (519.17, 456.78, 144) mm, rotated rx -180 ry 0 rz 160 deg; joints [0.702, 58.456, -5.667, -154.615, 55.549, 164.974]
  Set speed (16.7 mm/s)
  Call Extruder(164.54689)
  MoveL 8152 to (520.75, 457.52, 144) mm, rotated rx 180 ry 0 rz 160 deg; joints [0.789, 58.731, -6.207, -154.435, 55.332, 164.778]
  Set speed (16.7 mm/s)
  Call Extruder(170.31818)
  MoveL 8153 to (522.27, 458.29, 144) mm, rotated rx 180 ry 0 rz 160 deg; joints [0.881, 58.998, -6.731, -154.249, 55.124, 164.581]
  Set speed (16.7 mm/s)
  Call Extruder(176.29367)
  MoveL 8154 to (523.82, 459.16, 144) mm, rotated rx 180 ry 0 rz 160 deg; joints [0.983, 59.271, -7.268, -154.049, 54.915, 164.372]
  Set speed (16.7 mm/s)
  Call Extruder(182.07156)
  MoveL 8155 to (525.29, 460.05, 144) mm, rotated rx -180 ry 0 rz 160 deg; joints [1.087, 59.533, -7.781, -153.849, 54.717, 164.166]
  Set speed (16.7 mm/s)
  Call Extruder(187.80030)
  MoveL 8156 to (526.7, 460.98, 144) mm, rotated rx -180 ry 0 rz 160 deg; joints [1.196, 59.788, -8.282, -153.643, 54.527, 163.958]
  Set speed (16.7 mm/s)
  Call Extruder(193.73300)
  MoveL 8157 to (528.14, 462, 144) mm, rotated rx -180 ry 0 rz 160 deg; joints [1.315, 60.049, -8.793, -153.423, 54.336, 163.74]
  Call Extruder(199.77631)
  MoveL 8158 to (529.55, 463.09, 144) mm, rotated rx -180 ry 0 rz 160 deg; joints [1.442, 60.309, -9.303, -153.192, 54.148, 163.513]
  Set speed (16.7 mm/s)
  Call Extruder(205.55600)
  MoveL 8159 to (530.87, 464.19, 144) mm, rotated rx 180 ry 0 rz 160 deg; joints [1.568, 60.554, -9.782, -152.965, 53.975, 163.294]
  Set speed (16.7 mm/s)
  Call Extruder(211.42681)
  MoveL 8160 to (532.17, 465.35, 144) mm, rotated rx -180 ry 0 rz 160 deg; joints [1.702, 60.796, -10.258, -152.729, 53.807, 163.069]
  Set speed (16.7 mm/s)
  Call Extruder(217.37947)
  MoveL 8161 to (533.44, 466.57, 144) mm, rotated rx 180 ry 0 rz 160 deg; joints [1.843, 61.037, -10.729, -152.484, 53.643, 162.839]
  Call Extruder(220.52710)
  MoveL 8162 to (534.1, 467.24, 144) mm, rotated rx -180 ry 0 rz 160 deg; joints [1.919, 61.162, -10.973, -152.353, 53.56, 162.716]
  Call Extruder(223.75950)
  MoveL 8163 to (534.75, 467.94, 144) mm, rotated rx 180 ry 0 rz 160 deg; joints [1.999, 61.288, -11.221, -152.216, 53.477, 162.59]
  Set speed (16.7 mm/s)
  Call Extruder(227.02213)
  MoveL 8164 to (535.4, 468.66, 144) mm, rotated rx 180 ry 0 rz 160 deg; joints [2.081, 61.413, -11.466, -152.077, 53.396, 162.462]
  Set speed (16.7 mm/s)
  Call Extruder(230.27961)
  MoveL 8165 to (536.03, 469.39, 144) mm, rotated rx 180 ry 0 rz 160 deg; joints [2.165, 61.537, -11.707, -151.937, 53.317, 162.334]
  Set speed (16.7 mm/s)
  Call Extruder(233.58598)
  MoveL 8166 to (536.66, 470.14, 144) mm, rotated rx 180 ry 0 rz 160 deg; joints [2.25, 61.66, -11.948, -151.794, 53.239, 162.204]
  Set speed (16.7 mm/s)
  Call Extruder(236.86842)
  MoveL 8167 to (537.27, 470.9, 144) mm, rotated rx 180 ry 0 rz 160 deg; joints [2.337, 61.779, -12.182, -151.65, 53.165, 162.075]
  Set speed (16.7 mm/s)
  Call Extruder(240.05583)
  MoveL 8168 to (537.84, 471.65, 144) mm, rotated rx 180 ry 0 rz 160 deg; joints [2.422, 61.894, -12.405, -151.51, 53.095, 161.949]
  Set speed (16.7 mm/s)
  Call Extruder(242.83321)
  MoveL 8169 to (538.33, 472.31, 144) mm, rotated rx 180 ry 0 rz 160 deg; joints [2.498, 61.992, -12.596, -151.387, 53.037, 161.839]
  Set speed (16.7 mm/s)
  Call Extruder(248.70397)
  MoveL 8170 to (539.32, 473.75, 144) mm, rotated rx -180 ry 0 rz 160 deg; joints [2.66, 62.192, -12.988, -151.124, 52.92, 161.608]
  Set speed (16.7 mm/s)
  Call Extruder(253.07108)
  MoveL 8171 to (540.03, 474.83, 144) mm, rotated rx 180 ry 0 rz 160 deg; joints [2.783, 62.336, -13.27, -150.927, 52.838, 161.436]
  Set speed (16.7 mm/s)
  Call Extruder(256.43597)
  MoveL 8172 to (540.55, 475.68, 144) mm, rotated rx -180 ry 0 rz 160 deg; joints [2.88, 62.444, -13.481, -150.775, 52.779, 161.304]
  Call Extruder(259.59484)
  MoveL 8173 to (541.02, 476.49, 144) mm, rotated rx 180 ry 0 rz 160 deg; joints [2.971, 62.544, -13.675, -150.631, 52.726, 161.18]
  Set speed (16.7 mm/s)
  Call Extruder(264.99557)
  MoveL 8174 to (541.8, 477.89, 144) mm, rotated rx -180 ry 0 rz 160 deg; joints [3.129, 62.707, -13.994, -150.384, 52.642, 160.969]
  Set speed (16.7 mm/s)
  Call Extruder(269.46288)
  MoveL 8175 to (542.4, 479.07, 144) mm, rotated rx 180 ry 0 rz 160 deg; joints [3.262, 62.836, -14.247, -150.179, 52.578, 160.796]
  Set speed (16.7 mm/s)
  Call Extruder(274.66354)
  MoveL 8176 to (543.06, 480.46, 144) mm, rotated rx -180 ry 0 rz 160 deg; joints [3.419, 62.981, -14.529, -149.94, 52.511, 160.596]
  Set speed (16.7 mm/s)
  Call Extruder(279.29742)
  MoveL 8177 to (543.6, 481.72, 144) mm, rotated rx 180 ry 0 rz 160 deg; joints [3.562, 63.102, -14.764, -149.727, 52.459, 160.42]
  Set speed (16.7 mm/s)
  Call Extruder(282.60502)
  MoveL 8178 to (543.98, 482.63, 144) mm, rotated rx -180 ry 0 rz 160 deg; joints [3.664, 63.186, -14.929, -149.574, 52.424, 160.295]
  Set speed (16.7 mm/s)
  Call Extruder(285.82583)
  MoveL 8179 to (544.31, 483.52, 144) mm, rotated rx 180 ry 0 rz 160 deg; joints [3.764, 63.264, -15.08, -149.426, 52.395, 160.175]
  Set speed (16.7 mm/s)
  Call Extruder(289.09599)
  MoveL 8180 to (544.64, 484.43, 144) mm, rotated rx -180 ry 0 rz 160 deg; joints [3.867, 63.341, -15.23, -149.275, 52.367, 160.054]
  Set speed (16.7 mm/s)
  Call Extruder(295.62248)
  MoveL 8181 to (545.25, 486.27, 144) mm, rotated rx 180 ry 0 rz 160 deg; joints [4.074, 63.484, -15.511, -148.975, 52.321, 159.815]
  Set speed (16.7 mm/s)
  Call Extruder(301.92638)
  MoveL 8182 to (545.75, 488.07, 144) mm, rotated rx 180 ry 0 rz 160 deg; joints [4.277, 63.611, -15.757, -148.686, 52.288, 159.589]
  Set speed (16.7 mm/s)
  Call Extruder(305.42337)
  MoveL 8183 to (546, 489.07, 144) mm, rotated rx -180 ry 0 rz 160 deg; joints [4.391, 63.675, -15.882, -148.527, 52.276, 159.467]
  Set speed (16.7 mm/s)
  Call Extruder(308.56686)
  MoveL 8184 to (546.21, 489.98, 144) mm, rotated rx 180 ry 0 rz 160 deg; joints [4.493, 63.73, -15.991, -148.385, 52.267, 159.358]
  Set speed (16.7 mm/s)
  Call Extruder(315.06410)
  MoveL 8185 to (546.58, 491.87, 144) mm, rotated rx 180 ry 0 rz 160 deg; joints [4.707, 63.834, -16.193, -148.092, 52.259, 159.137]
  Call Extruder(321.73361)
  MoveL 8186 to (546.88, 493.82, 144) mm, rotated rx 180 ry 0 rz 160 deg; joints [4.928, 63.927, -16.374, -147.795, 52.263, 158.918]
  Set speed (16.7 mm/s)
  Call Extruder(328.32720)
  MoveL 8187 to (547.09, 495.77, 144) mm, rotated rx -180 ry 0 rz 160 deg; joints [5.148, 64.004, -16.525, -147.504, 52.281, 158.71]
  Set speed (16.7 mm/s)
  Call Extruder(334.75997)
  MoveL 8188 to (547.23, 497.67, 144) mm, rotated rx -180 ry 0 rz 160 deg; joints [5.365, 64.066, -16.646, -147.225, 52.31, 158.514]
  Call Extruder(341.27424)
  MoveL 8189 to (547.28, 499.6, 144) mm, rotated rx 180 ry 0 rz 160 deg; joints [5.585, 64.115, -16.74, -146.947, 52.353, 158.324]
  Set speed (16.7 mm/s)
  Call Extruder(347.64673)
  MoveL 8190 to (547.26, 501.49, 144) mm, rotated rx 180 ry 0 rz 160 deg; joints [5.801, 64.148, -16.806, -146.68, 52.406, 158.148]
  Set speed (16.7 mm/s)
  Call Extruder(354.30311)
  MoveL 8191 to (547.16, 503.46, 144) mm, rotated rx -180 ry 0 rz 160 deg; joints [6.028, 64.169, -16.845, -146.407, 52.475, 157.973]
  Set speed (16.7 mm/s)
  Call Extruder(360.75590)
  MoveL 8192 to (546.98, 505.37, 144) mm, rotated rx 180 ry 0 rz 160 deg; joints [6.247, 64.174, -16.855, -146.149, 52.554, 157.813]
  Set speed (16.7 mm/s)
  Call Extruder(367.45380)
  MoveL 8193 to (546.71, 507.33, 144) mm, rotated rx 180 ry 0 rz 160 deg; joints [6.475, 64.164, -16.836, -145.887, 52.647, 157.658]
  Set speed (16.7 mm/s)
  Call Extruder(373.86879)
  MoveL 8194 to (546.38, 509.21, 144) mm, rotated rx 180 ry 0 rz 160 deg; joints [6.693, 64.141, -16.791, -145.643, 52.749, 157.521]
  Set speed (16.7 mm/s)
  Call Extruder(380.50313)
  MoveL 8195 to (545.96, 511.13, 144) mm, rotated rx -180 ry 0 rz 160 deg; joints [6.918, 64.102, -16.715, -145.398, 52.865, 157.389]
  Call Extruder(387.12137)
  MoveL 8196 to (545.46, 513.03, 144) mm, rotated rx 180 ry 0 rz 160 deg; joints [7.141, 64.049, -16.611, -145.162, 52.993, 157.269]
  Set speed (16.7 mm/s)
  Call Extruder(393.33248)
  MoveL 8197 to (544.91, 514.79, 144) mm, rotated rx 180 ry 0 rz 160 deg; joints [7.35, 63.985, -16.487, -144.947, 53.123, 157.168]
  Set speed (16.7 mm/s)
  Call Extruder(400.13159)
  MoveL 8198 to (544.24, 516.69, 144) mm, rotated rx 180 ry 0 rz 160 deg; joints [7.577, 63.901, -16.323, -144.721, 53.277, 157.069]
  Set speed (16.7 mm/s)
  Call Extruder(406.58515)
  MoveL 8199 to (543.53, 518.47, 144) mm, rotated rx 180 ry 0 rz 160 deg; joints [7.791, 63.807, -16.141, -144.513, 53.432, 156.987]
  Call Extruder(412.94916)
  MoveL 8200 to (542.76, 520.19, 144) mm, rotated rx 180 ry 0 rz 160 deg; joints [7.999, 63.702, -15.935, -144.318, 53.596, 156.917]
  Set speed (16.7 mm/s)
  Call Extruder(416.21127)
  MoveL 8201 to (542.33, 521.06, 144) mm, rotated rx 180 ry 0 rz 160 deg; joints [8.106, 63.642, -15.819, -144.221, 53.683, 156.886]
  Set speed (16.7 mm/s)
  Call Extruder(419.42711)
  MoveL 8202 to (541.9, 521.91, 144) mm, rotated rx -180 ry 0 rz 160 deg; joints [8.21, 63.581, -15.7, -144.127, 53.771, 156.858]
  Set speed (16.7 mm/s)
  Call Extruder(422.71750)
  MoveL 8203 to (541.44, 522.77, 144) mm, rotated rx -180 ry 0 rz 160 deg; joints [8.316, 63.515, -15.571, -144.033, 53.864, 156.832]
  Set speed (16.7 mm/s)
  Call Extruder(425.97225)
  MoveL 8204 to (540.97, 523.61, 144) mm, rotated rx 180 ry 0 rz 160 deg; joints [8.42, 63.447, -15.438, -143.942, 53.958, 156.81]
  Set speed (16.7 mm/s)
  Call Extruder(429.33916)
  MoveL 8205 to (540.46, 524.47, 144) mm, rotated rx 180 ry 0 rz 160 deg; joints [8.527, 63.372, -15.293, -143.851, 54.057, 156.79]
  Set speed (16.7 mm/s)
  Call Extruder(432.49699)
  MoveL 8206 to (539.97, 525.27, 144) mm, rotated rx 180 ry 0 rz 160 deg; joints [8.627, 63.3, -15.151, -143.767, 54.152, 156.774]
  Set speed (16.7 mm/s)
  Call Extruder(435.76693)
  MoveL 8207 to (539.44, 526.08, 144) mm, rotated rx -180 ry 0 rz 160 deg; joints [8.729, 63.222, -14.998, -143.683, 54.252, 156.761]
  Set speed (16.7 mm/s)
  Call Extruder(439.07001)
  MoveL 8208 to (538.89, 526.89, 144) mm, rotated rx 180 ry 0 rz 160 deg; joints [8.832, 63.139, -14.838, -143.6, 54.356, 156.75]
  Set speed (16.7 mm/s)
  Call Extruder(442.26197)
  MoveL 8209 to (538.35, 527.67, 144) mm, rotated rx 180 ry 0 rz 160 deg; joints [8.93, 63.058, -14.678, -143.522, 54.457, 156.742]
  Set speed (16.7 mm/s)
  Call Extruder(445.59686)
  MoveL 8210 to (537.76, 528.46, 144) mm, rotated rx -180 ry 0 rz 160 deg; joints [9.032, 62.969, -14.505, -143.443, 54.565, 156.737]
  Set speed (16.7 mm/s)
  Call Extruder(449.62206)
  MoveL 8211 to (537.03, 529.41, 144) mm, rotated rx -180 ry 0 rz 160 deg; joints [9.154, 62.857, -14.287, -143.351, 54.699, 156.735]
  Set speed (16.7 mm/s)
  Call Extruder(455.26353)
  MoveL 8212 to (535.96, 530.7, 144) mm, rotated rx -180 ry 0 rz 160 deg; joints [9.322, 62.693, -13.967, -143.227, 54.89, 156.74]
  Set speed (16.7 mm/s)
  Call Extruder(458.62132)
  MoveL 8213 to (535.31, 531.45, 144) mm, rotated rx 180 ry 0 rz 160 deg; joints [9.421, 62.592, -13.77, -143.157, 55.007, 156.747]
  Set speed (16.7 mm/s)
  Call Extruder(461.91373)
  MoveL 8214 to (534.65, 532.17, 144) mm, rotated rx -180 ry 0 rz 160 deg; joints [9.517, 62.49, -13.57, -143.091, 55.122, 156.757]
  Call Extruder(465.22286)
  MoveL 8215 to (533.98, 532.88, 144) mm, rotated rx -180 ry 0 rz 160 deg; joints [9.612, 62.385, -13.365, -143.026, 55.24, 156.769]
  Set speed (16.7 mm/s)
  Call Extruder(468.37038)
  MoveL 8216 to (533.32, 533.55, 144) mm, rotated rx 180 ry 0 rz 160 deg; joints [9.701, 62.283, -13.165, -142.967, 55.353, 156.784]
  Call Extruder(471.66596)
  MoveL 8217 to (532.62, 534.23, 144) mm, rotated rx -180 ry 0 rz 160 deg; joints [9.794, 62.173, -12.951, -142.907, 55.473, 156.802]
  Set speed (16.7 mm/s)
  Call Extruder(474.91865)
  MoveL 8218 to (531.92, 534.88, 144) mm, rotated rx -180 ry 0 rz 160 deg; joints [9.884, 62.062, -12.734, -142.85, 55.593, 156.823]
  Call Extruder(478.26967)
  MoveL 8219 to (531.18, 535.55, 144) mm, rotated rx 180 ry 0 rz 160 deg; joints [9.975, 61.946, -12.506, -142.794, 55.717, 156.847]
  Set speed (16.7 mm/s)
  Call Extruder(481.00430)
  MoveL 8220 to (530.56, 536.08, 144) mm, rotated rx 180 ry 0 rz 160 deg; joints [10.049, 61.849, -12.317, -142.75, 55.82, 156.868]
  Set speed (16.7 mm/s)
  Call Extruder(486.91722)
  MoveL 8221 to (529.21, 537.19, 144) mm, rotated rx -180 ry 0 rz 160 deg; joints [10.206, 61.634, -11.897, -142.66, 56.045, 156.921]
  Set speed (16.7 mm/s)
  Call Extruder(489.73769)
  MoveL 8222 to (528.54, 537.7, 144) mm, rotated rx 180 ry 0 rz 160 deg; joints [10.279, 61.529, -11.692, -142.62, 56.153, 156.949]
  Set speed (16.7 mm/s)
  Call Extruder(491.95645)
  MoveL 8223 to (528.02, 538.09, 144) mm, rotated rx -180 ry 0 rz 160 deg; joints [10.336, 61.445, -11.528, -142.59, 56.239, 156.972]
  Set speed (16.7 mm/s)
  Call Extruder(497.67641)
  MoveL 8224 to (526.63, 539.07, 144) mm, rotated rx -180 ry 0 rz 160 deg; joints [10.479, 61.224, -11.096, -142.516, 56.463, 157.039]
  Set speed (16.7 mm/s)
  Call Extruder(501.00062)
  MoveL 8225 to (525.81, 539.62, 144) mm, rotated rx -180 ry 0 rz 160 deg; joints [10.561, 61.093, -10.839, -142.477, 56.594, 157.081]
  Set speed (16.7 mm/s)
  Call Extruder(504.32550)
  MoveL 8226 to (524.98, 540.15, 144) mm, rotated rx -180 ry 0 rz 160 deg; joints [10.641, 60.961, -10.58, -142.44, 56.726, 157.125]
  Set speed (16.7 mm/s)
  Call Extruder(507.55375)
  MoveL 8227 to (524.16, 540.64, 144) mm, rotated rx -180 ry 0 rz 160 deg; joints [10.717, 60.83, -10.323, -142.406, 56.855, 157.17]
  Set speed (16.7 mm/s)
  Call Extruder(510.79905)
  MoveL 8228 to (523.33, 541.13, 144) mm, rotated rx 180 ry 0 rz 160 deg; joints [10.792, 60.697, -10.063, -142.375, 56.985, 157.218]
  Call Extruder(514.04278)
  MoveL 8229 to (522.49, 541.59, 144) mm, rotated rx -180 ry 0 rz 160 deg; joints [10.865, 60.562, -9.799, -142.345, 57.115, 157.268]
  Call Extruder(517.31560)
  MoveL 8230 to (521.63, 542.05, 144) mm, rotated rx 180 ry 0 rz 160 deg; joints [10.937, 60.424, -9.529, -142.318, 57.248, 157.321]
  Call Extruder(520.60439)
  MoveL 8231 to (520.76, 542.48, 144) mm, rotated rx -180 ry 0 rz 160 deg; joints [11.009, 60.284, -9.255, -142.292, 57.382, 157.377]
  Set speed (16.7 mm/s)
  Call Extruder(523.78840)
  MoveL 8232 to (519.91, 542.89, 144) mm, rotated rx 180 ry 0 rz 160 deg; joints [11.076, 60.148, -8.987, -142.27, 57.511, 157.432]
  Set speed (16.7 mm/s)
  Call Extruder(527.18940)
  MoveL 8233 to (518.99, 543.3, 144) mm, rotated rx 180 ry 0 rz 160 deg; joints [11.146, 60, -8.697, -142.249, 57.65, 157.495]
  Set speed (16.7 mm/s)
  Call Extruder(530.34801)
  MoveL 8234 to (518.13, 543.67, 144) mm, rotated rx 180 ry 0 rz 160 deg; joints [11.209, 59.861, -8.426, -142.23, 57.78, 157.553]
  Set speed (16.7 mm/s)
  Call Extruder(536.76135)
  MoveL 8235 to (516.36, 544.36, 144) mm, rotated rx 180 ry 0 rz 160 deg; joints [11.333, 59.576, -7.867, -142.201, 58.043, 157.68]
  Set speed (16.7 mm/s)
  Call Extruder(543.35870)
  MoveL 8236 to (514.51, 545, 144) mm, rotated rx -180 ry 0 rz 160 deg; joints [11.453, 59.279, -7.283, -142.18, 58.315, 157.818]
  Set speed (16.7 mm/s)
  Call Extruder(548.06506)
  MoveL 8237 to (513.18, 545.41, 144) mm, rotated rx -180 ry 0 rz 160 deg; joints [11.533, 59.064, -6.861, -142.17, 58.509, 157.921]
  Call Extruder(550.10969)
  MoveL 8238 to (512.6, 545.58, 144) mm, rotated rx 180 ry 0 rz 160 deg; joints [11.567, 58.97, -6.677, -142.167, 58.593, 157.967]
  Set speed (16.7 mm/s)
  Call Extruder(552.73172)
  MoveL 8239 to (511.85, 545.77, 144) mm, rotated rx 180 ry 0 rz 160 deg; joints [11.609, 58.849, -6.438, -142.165, 58.701, 158.027]
  Set speed (16.7 mm/s)
  Call Extruder(556.54276)
  MoveL 8240 to (510.75, 546.05, 144) mm, rotated rx 180 ry 0 rz 160 deg; joints [11.668, 58.672, -6.091, -142.164, 58.858, 158.116]
  Set speed (16.7 mm/s)
  Call Extruder(563.09508)
  MoveL 8241 to (508.85, 546.45, 144) mm, rotated rx 180 ry 0 rz 160 deg; joints [11.764, 58.365, -5.488, -142.17, 59.127, 158.275]
  Set speed (16.7 mm/s)
  Call Extruder(569.49231)
  MoveL 8242 to (506.98, 546.77, 144) mm, rotated rx 180 ry 0 rz 160 deg; joints [11.849, 58.063, -4.894, -142.185, 59.389, 158.436]
  Set speed (16.7 mm/s)
  Call Extruder(576.10662)
  MoveL 8243 to (505.04, 547.01, 144) mm, rotated rx 180 ry 0 rz 160 deg; joints [11.928, 57.748, -4.275, -142.209, 59.658, 158.609]
  Set speed (16.7 mm/s)
  Call Extruder(582.69679)
  MoveL 8244 to (503.09, 547.18, 144) mm, rotated rx -180 ry 0 rz 160 deg; joints [11.998, 57.433, -3.655, -142.242, 59.925, 158.787]
  Set speed (16.7 mm/s)
  Call Extruder(589.26684)
  MoveL 8245 to (501.14, 547.27, 144) mm, rotated rx 180 ry 0 rz 160 deg; joints [12.059, 57.118, -3.034, -142.284, 60.189, 158.97]
  Set speed (16.7 mm/s)
  Call Extruder(595.69097)
  MoveL 8246 to (499.24, 547.28, 144) mm, rotated rx 180 ry 0 rz 160 deg; joints [12.11, 56.809, -2.426, -142.334, 60.444, 159.154]
  Set speed (10.0 mm/s)
  MoveL 8247 to (499.24, 547.28, 148) mm, rotated rx -180 ry 0 rz 160 deg; joints [12.11, 56.23, -2.27, -142.186, 60.109, 158.856]
  Set speed (120.0 mm/s)
  MoveL 8248 to (499.22, 545.71, 148) mm, rotated rx 180 ry 0 rz 160 deg; joints [11.919, 56.173, -2.158, -142.411, 60.084, 158.997]
  Set speed (16.8 mm/s)
  Call Extruder(602.02863)
  MoveL 8249 to (497.33, 545.64, 148) mm, rotated rx 180 ry 0 rz 160 deg; joints [11.959, 55.865, -1.554, -142.47, 60.332, 159.183]
  Set speed (16.8 mm/s)
  Call Extruder(608.32297)
  MoveL 8250 to (495.46, 545.5, 148) mm, rotated rx -180 ry 0 rz 160 deg; joints [11.99, 55.559, -0.955, -142.538, 60.576, 159.372]
  Set speed (16.8 mm/s)
  Call Extruder(614.36738)
  MoveL 8251 to (493.67, 545.28, 148) mm, rotated rx 180 ry 0 rz 160 deg; joints [12.011, 55.266, -0.381, -142.612, 60.807, 159.557]
  Call Extruder(620.61667)
  MoveL 8252 to (491.83, 544.98, 148) mm, rotated rx 180 ry 0 rz 160 deg; joints [12.022, 54.964, 0.21, -142.698, 61.041, 159.752]
  Call Extruder(627.07477)
  MoveL 8253 to (489.94, 544.6, 148) mm, rotated rx 180 ry 0 rz 160 deg; joints [12.025, 54.655, 0.818, -142.794, 61.279, 159.957]
  Set speed (16.8 mm/s)
  Call Extruder(633.05769)
  MoveL 8254 to (488.21, 544.17, 148) mm, rotated rx 180 ry 0 rz 160 deg; joints [12.017, 54.37, 1.377, -142.893, 61.495, 160.149]
  Call Extruder(639.28728)
  MoveL 8255 to (486.43, 543.66, 148) mm, rotated rx -180 ry 0 rz 160 deg; joints [12, 54.076, 1.955, -143.003, 61.716, 160.352]
  Set speed (16.8 mm/s)
  Call Extruder(645.56628)
  MoveL 8256 to (484.65, 543.07, 148) mm, rotated rx -180 ry 0 rz 160 deg; joints [11.973, 53.782, 2.531, -143.123, 61.933, 160.558]
  Set speed (16.8 mm/s)
  Call Extruder(647.27011)
  MoveL 8257 to (484.17, 542.89, 148) mm, rotated rx 180 ry 0 rz 160 deg; joints [11.964, 53.704, 2.686, -143.157, 61.991, 160.615]
  Set speed (16.8 mm/s)
  Call Extruder(652.22037)
  MoveL 8258 to (482.8, 542.36, 148) mm, rotated rx -180 ry 0 rz 160 deg; joints [11.934, 53.476, 3.133, -143.26, 62.156, 160.779]
  Set speed (16.8 mm/s)
  Call Extruder(658.18745)
  MoveL 8259 to (481.16, 541.66, 148) mm, rotated rx -180 ry 0 rz 160 deg; joints [11.888, 53.204, 3.667, -143.39, 62.352, 160.979]
  Set speed (16.8 mm/s)
  Call Extruder(662.48076)
  MoveL 8260 to (480, 541.12, 148) mm, rotated rx -180 ry 0 rz 160 deg; joints [11.851, 53.011, 4.048, -143.489, 62.49, 161.123]
  Set speed (16.8 mm/s)
  Call Extruder(666.15340)
  MoveL 8261 to (479.02, 540.63, 148) mm, rotated rx -180 ry 0 rz 160 deg; joints [11.814, 52.848, 4.369, -143.577, 62.605, 161.247]
  Set speed (16.8 mm/s)
  Call Extruder(670.75102)
  MoveL 8262 to (477.82, 539.98, 148) mm, rotated rx 180 ry 0 rz 160 deg; joints [11.763, 52.646, 4.766, -143.691, 62.746, 161.402]
  Set speed (16.8 mm/s)
  Call Extruder(674.71276)
  MoveL 8263 to (476.79, 539.39, 148) mm, rotated rx 180 ry 0 rz 160 deg; joints [11.715, 52.474, 5.104, -143.793, 62.865, 161.536]
  Set speed (16.8 mm/s)
  Call Extruder(680.12982)
  MoveL 8264 to (475.42, 538.54, 148) mm, rotated rx 180 ry 0 rz 160 deg; joints [11.642, 52.243, 5.56, -143.938, 63.023, 161.72]
  Set speed (16.8 mm/s)
  Call Extruder(683.26715)
  MoveL 8265 to (474.63, 538.03, 148) mm, rotated rx -180 ry 0 rz 160 deg; joints [11.597, 52.111, 5.82, -144.024, 63.113, 161.826]
  Call Extruder(686.44625)
  MoveL 8266 to (473.85, 537.5, 148) mm, rotated rx -180 ry 0 rz 160 deg; joints [11.548, 51.978, 6.081, -144.114, 63.202, 161.934]
  Set speed (16.8 mm/s)
  Call Extruder(689.71478)
  MoveL 8267 to (473.05, 536.93, 148) mm, rotated rx 180 ry 0 rz 160 deg; joints [11.496, 51.844, 6.346, -144.209, 63.291, 162.045]
  Set speed (16.8 mm/s)
  Call Extruder(692.75075)
  MoveL 8268 to (472.33, 536.39, 148) mm, rotated rx 180 ry 0 rz 160 deg; joints [11.444, 51.72, 6.589, -144.299, 63.373, 162.148]
  Set speed (16.8 mm/s)
  Call Extruder(695.78179)
  MoveL 8269 to (471.61, 535.84, 148) mm, rotated rx 180 ry 0 rz 160 deg; joints [11.391, 51.599, 6.829, -144.39, 63.452, 162.25]
  Set speed (16.8 mm/s)
  Call Extruder(698.99499)
  MoveL 8270 to (470.87, 535.24, 148) mm, rotated rx 180 ry 0 rz 160 deg; joints [11.331, 51.472, 7.079, -144.489, 63.535, 162.359]
  Call Extruder(702.15092)
  MoveL 8271 to (470.15, 534.63, 148) mm, rotated rx -180 ry 0 rz 160 deg; joints [11.271, 51.348, 7.323, -144.588, 63.614, 162.465]
  Set speed (16.8 mm/s)
  Call Extruder(705.23673)
  MoveL 8272 to (469.46, 534.02, 148) mm, rotated rx 180 ry 0 rz 160 deg; joints [11.209, 51.23, 7.557, -144.687, 63.69, 162.569]
  Call Extruder(708.39502)
  MoveL 8273 to (468.76, 533.38, 148) mm, rotated rx -180 ry 0 rz 160 deg; joints [11.143, 51.11, 7.793, -144.791, 63.765, 162.675]
  Set speed (16.8 mm/s)
  Call Extruder(711.24192)
  MoveL 8274 to (468.15, 532.8, 148) mm, rotated rx -180 ry 0 rz 160 deg; joints [11.082, 51.004, 8.002, -144.885, 63.831, 162.77]
  Call Extruder(714.66650)
  MoveL 8275 to (467.42, 532.08, 148) mm, rotated rx -180 ry 0 rz 160 deg; joints [11.005, 50.878, 8.25, -145.001, 63.909, 162.884]
  Set speed (16.8 mm/s)
  Call Extruder(717.77496)
  MoveL 8276 to (466.78, 531.41, 148) mm, rotated rx 180 ry 0 rz 160 deg; joints [10.933, 50.766, 8.471, -145.108, 63.977, 162.987]
  Set speed (16.8 mm/s)
  Call Extruder(720.93700)
  MoveL 8277 to (466.14, 530.72, 148) mm, rotated rx 180 ry 0 rz 160 deg; joints [10.857, 50.655, 8.692, -145.219, 64.044, 163.092]
  Set speed (16.8 mm/s)
  Call Extruder(724.04945)
  MoveL 8278 to (465.52, 530.02, 148) mm, rotated rx -180 ry 0 rz 160 deg; joints [10.781, 50.547, 8.905, -145.33, 64.109, 163.194]
  Set speed (16.8 mm/s)
  Call Extruder(727.21233)
  MoveL 8279 to (464.91, 529.31, 148) mm, rotated rx 180 ry 0 rz 160 deg; joints [10.701, 50.439, 9.119, -145.444, 64.172, 163.298]
  Set speed (16.8 mm/s)
  Call Extruder(730.35159)
  MoveL 8280 to (464.32, 528.58, 148) mm, rotated rx 180 ry 0 rz 160 deg; joints [10.618, 50.334, 9.325, -145.559, 64.233, 163.4]
  Set speed (16.8 mm/s)
  Call Extruder(733.65144)
  MoveL 8281 to (463.71, 527.81, 148) mm, rotated rx -180 ry 0 rz 160 deg; joints [10.53, 50.226, 9.539, -145.682, 64.295, 163.507]
  Set speed (16.8 mm/s)
  Call Extruder(736.62749)
  MoveL 8282 to (463.18, 527.1, 148) mm, rotated rx -180 ry 0 rz 160 deg; joints [10.448, 50.131, 9.727, -145.795, 64.348, 163.603]
  Set speed (16.8 mm/s)
  Call Extruder(739.89370)
  MoveL 8283 to (462.61, 526.31, 148) mm, rotated rx -180 ry 0 rz 160 deg; joints [10.355, 50.029, 9.928, -145.92, 64.405, 163.708]
  Call Extruder(742.85240)
  MoveL 8284 to (462.11, 525.58, 148) mm, rotated rx 180 ry 0 rz 160 deg; joints [10.27, 49.938, 10.107, -146.035, 64.454, 163.802]
  Set speed (16.8 mm/s)
  Call Extruder(748.68337)
  MoveL 8285 to (461.16, 524.12, 148) mm, rotated rx -180 ry 0 rz 160 deg; joints [10.096, 49.766, 10.448, -146.264, 64.546, 163.985]
  Set speed (16.8 mm/s)
  Call Extruder(752.31985)
  MoveL 8286 to (460.6, 523.19, 148) mm, rotated rx 180 ry 0 rz 160 deg; joints [9.983, 49.664, 10.651, -146.411, 64.598, 164.098]
  Set speed (16.8 mm/s)
  Call Extruder(755.39641)
  MoveL 8287 to (460.14, 522.4, 148) mm, rotated rx 180 ry 0 rz 160 deg; joints [9.886, 49.579, 10.819, -146.536, 64.641, 164.193]
  Set speed (16.8 mm/s)
  Call Extruder(758.58187)
  MoveL 8288 to (459.69, 521.57, 148) mm, rotated rx -180 ry 0 rz 160 deg; joints [9.784, 49.494, 10.987, -146.667, 64.683, 164.291]
  Set speed (16.8 mm/s)
  Call Extruder(761.64823)
  MoveL 8289 to (459.26, 520.76, 148) mm, rotated rx 180 ry 0 rz 160 deg; joints [9.684, 49.414, 11.145, -146.794, 64.721, 164.384]
  Set speed (16.8 mm/s)
  Call Extruder(764.84551)
  MoveL 8290 to (458.84, 519.9, 148) mm, rotated rx 180 ry 0 rz 160 deg; joints [9.577, 49.334, 11.303, -146.928, 64.758, 164.48]
  Set speed (16.8 mm/s)
  Call Extruder(768.15045)
  MoveL 8291 to (458.42, 519.01, 148) mm, rotated rx 180 ry 0 rz 160 deg; joints [9.464, 49.254, 11.462, -147.068, 64.794, 164.578]
  Set speed (16.8 mm/s)
  Call Extruder(771.12132)
  MoveL 8292 to (458.06, 518.2, 148) mm, rotated rx 180 ry 0 rz 160 deg; joints [9.362, 49.184, 11.6, -147.194, 64.824, 164.666]
  Set speed (16.8 mm/s)
  Call Extruder(778.35834)
  MoveL 8293 to (457.24, 516.2, 148) mm, rotated rx -180 ry 0 rz 160 deg; joints [9.106, 49.023, 11.919, -147.507, 64.89, 164.875]
  Set speed (16.8 mm/s)
  Call Extruder(783.59445)
  MoveL 8294 to (456.72, 514.73, 148) mm, rotated rx -180 ry 0 rz 160 deg; joints [8.915, 48.917, 12.128, -147.736, 64.928, 165.023]
  Set speed (16.8 mm/s)
  Call Extruder(786.97143)
  MoveL 8295 to (456.41, 513.78, 148) mm, rotated rx -180 ry 0 rz 160 deg; joints [8.79, 48.852, 12.257, -147.886, 64.949, 165.117]
  Call Extruder(790.08897)
  MoveL 8296 to (456.13, 512.89, 148) mm, rotated rx 180 ry 0 rz 160 deg; joints [8.674, 48.795, 12.371, -148.024, 64.967, 165.203]
  Set speed (16.8 mm/s)
  Call Extruder(796.14716)
  MoveL 8297 to (455.66, 511.15, 148) mm, rotated rx 180 ry 0 rz 160 deg; joints [8.442, 48.692, 12.575, -148.296, 64.995, 165.366]
  Set speed (16.8 mm/s)
  Call Extruder(799.51200)
  MoveL 8298 to (455.43, 510.17, 148) mm, rotated rx 180 ry 0 rz 160 deg; joints [8.312, 48.64, 12.678, -148.448, 65.005, 165.455]
  Call Extruder(802.68147)
  MoveL 8299 to (455.23, 509.25, 148) mm, rotated rx -180 ry 0 rz 160 deg; joints [8.188, 48.592, 12.772, -148.591, 65.014, 165.537]
  Set speed (16.8 mm/s)
  Call Extruder(808.86782)
  MoveL 8300 to (454.89, 507.43, 148) mm, rotated rx -180 ry 0 rz 160 deg; joints [7.943, 48.51, 12.936, -148.873, 65.022, 165.695]
  Set speed (16.8 mm/s)
  Call Extruder(815.14495)
  MoveL 8301 to (454.62, 505.58, 148) mm, rotated rx 180 ry 0 rz 160 deg; joints [7.69, 48.437, 13.081, -149.16, 65.022, 165.849]
  Set speed (16.8 mm/s)
  Call Extruder(821.50529)
  MoveL 8302 to (454.43, 503.69, 148) mm, rotated rx 180 ry 0 rz 160 deg; joints [7.43, 48.375, 13.203, -149.453, 65.011, 166.001]
  Set speed (16.8 mm/s)
  Call Extruder(828.76287)
  MoveL 8303 to (454.3, 501.53, 148) mm, rotated rx 180 ry 0 rz 160 deg; joints [7.131, 48.318, 13.315, -149.786, 64.987, 166.167]
  Call Extruder(833.72728)
  MoveL 8304 to (454.28, 500.05, 148) mm, rotated rx 180 ry 0 rz 160 deg; joints [6.925, 48.29, 13.372, -150.014, 64.962, 166.277]
  Call Extruder(839.65817)
  MoveL 8305 to (454.31, 498.29, 148) mm, rotated rx 180 ry 0 rz 160 deg; joints [6.676, 48.265, 13.42, -150.286, 64.924, 166.403]
  Set speed (16.8 mm/s)
  Call Extruder(845.28378)
  MoveL 8306 to (454.41, 496.61, 148) mm, rotated rx 180 ry 0 rz 160 deg; joints [6.44, 48.252, 13.448, -150.543, 64.88, 166.517]
  Set speed (16.8 mm/s)
  Call Extruder(850.71566)
  MoveL 8307 to (454.56, 495, 148) mm, rotated rx -180 ry 0 rz 160 deg; joints [6.212, 48.247, 13.456, -150.789, 64.831, 166.624]
  Set speed (16.8 mm/s)
  Call Extruder(856.56423)
  MoveL 8308 to (454.78, 493.27, 148) mm, rotated rx -180 ry 0 rz 160 deg; joints [5.966, 48.253, 13.445, -151.053, 64.77, 166.734]
  Set speed (16.8 mm/s)
  Call Extruder(862.16975)
  MoveL 8309 to (455.06, 491.62, 148) mm, rotated rx 180 ry 0 rz 160 deg; joints [5.73, 48.268, 13.415, -151.303, 64.703, 166.834]
  Set speed (16.8 mm/s)
  Call Extruder(867.84521)
  MoveL 8310 to (455.4, 489.96, 148) mm, rotated rx 180 ry 0 rz 160 deg; joints [5.493, 48.293, 13.366, -151.553, 64.628, 166.931]
  Call Extruder(873.48954)
  MoveL 8311 to (455.8, 488.32, 148) mm, rotated rx -180 ry 0 rz 160 deg; joints [5.258, 48.327, 13.298, -151.798, 64.545, 167.021]
  Call Extruder(879.14814)
  MoveL 8312 to (456.26, 486.7, 148) mm, rotated rx 180 ry 0 rz 160 deg; joints [5.025, 48.371, 13.21, -152.041, 64.454, 167.107]
  Call Extruder(884.87560)
  MoveL 8313 to (456.79, 485.08, 148) mm, rotated rx 180 ry 0 rz 160 deg; joints [4.791, 48.425, 13.103, -152.282, 64.355, 167.189]
  Set speed (16.8 mm/s)
  Call Extruder(890.14060)
  MoveL 8314 to (457.33, 483.6, 148) mm, rotated rx 180 ry 0 rz 160 deg; joints [4.578, 48.484, 12.986, -152.499, 64.257, 167.259]
  Set speed (16.8 mm/s)
  Call Extruder(896.09860)
  MoveL 8315 to (457.99, 481.96, 148) mm, rotated rx 180 ry 0 rz 160 deg; joints [4.341, 48.56, 12.836, -152.74, 64.138, 167.333]
  Set speed (16.8 mm/s)
  Call Extruder(901.49385)
  MoveL 8316 to (458.65, 480.49, 148) mm, rotated rx 180 ry 0 rz 160 deg; joints [4.129, 48.638, 12.682, -152.953, 64.024, 167.395]
  Set speed (16.8 mm/s)
  Call Extruder(907.35790)
  MoveL 8317 to (459.43, 478.92, 148) mm, rotated rx 180 ry 0 rz 160 deg; joints [3.902, 48.732, 12.496, -153.179, 63.893, 167.457]
  Set speed (16.8 mm/s)
  Call Extruder(913.02560)
  MoveL 8318 to (460.24, 477.44, 148) mm, rotated rx -180 ry 0 rz 160 deg; joints [3.688, 48.832, 12.297, -153.39, 63.758, 167.51]
  Set speed (16.8 mm/s)
  Call Extruder(918.43084)
  MoveL 8319 to (461.06, 476.05, 148) mm, rotated rx 180 ry 0 rz 160 deg; joints [3.487, 48.936, 12.092, -153.586, 63.624, 167.556]
  Set speed (16.8 mm/s)
  Call Extruder(924.28616)
  MoveL 8320 to (462, 474.58, 148) mm, rotated rx -180 ry 0 rz 160 deg; joints [3.275, 49.057, 11.851, -153.791, 63.471, 167.6]
  Set speed (16.8 mm/s)
  Call Extruder(929.93412)
  MoveL 8321 to (462.96, 473.2, 148) mm, rotated rx -180 ry 0 rz 160 deg; joints [3.076, 49.184, 11.601, -153.981, 63.318, 167.637]
  Set speed (16.8 mm/s)
  Call Extruder(935.60713)
  MoveL 8322 to (463.98, 471.84, 148) mm, rotated rx -180 ry 0 rz 160 deg; joints [2.881, 49.319, 11.333, -154.165, 63.157, 167.668]
  Set speed (16.8 mm/s)
  Call Extruder(941.20349)
  MoveL 8323 to (465.03, 470.55, 148) mm, rotated rx -180 ry 0 rz 160 deg; joints [2.695, 49.46, 11.053, -154.338, 62.992, 167.692]
  Call Extruder(946.83956)
  MoveL 8324 to (466.14, 469.28, 148) mm, rotated rx 180 ry 0 rz 160 deg; joints [2.514, 49.611, 10.755, -154.505, 62.821, 167.712]
  Set speed (16.8 mm/s)
  Call Extruder(952.59232)
  MoveL 8325 to (467.32, 468.03, 148) mm, rotated rx 180 ry 0 rz 160 deg; joints [2.335, 49.773, 10.434, -154.666, 62.64, 167.725]
  Set speed (16.8 mm/s)
  Call Extruder(958.14700)
  MoveL 8326 to (468.5, 466.87, 148) mm, rotated rx 180 ry 0 rz 160 deg; joints [2.169, 49.937, 10.11, -154.813, 62.459, 167.732]
  Set speed (16.8 mm/s)
  Call Extruder(963.78148)
  MoveL 8327 to (469.74, 465.73, 148) mm, rotated rx 180 ry 0 rz 160 deg; joints [2.008, 50.111, 9.767, -154.953, 62.271, 167.733]
  Call Extruder(969.48605)
  MoveL 8328 to (471.03, 464.63, 148) mm, rotated rx 180 ry 0 rz 160 deg; joints [1.852, 50.294, 9.404, -155.086, 62.076, 167.728]
  Set speed (16.8 mm/s)
  Call Extruder(975.06459)
  MoveL 8329 to (472.34, 463.6, 148) mm, rotated rx -180 ry 0 rz 160 deg; joints [1.706, 50.48, 9.036, -155.207, 61.88, 167.718]
  Set speed (16.8 mm/s)
  Call Extruder(980.70130)
  MoveL 8330 to (473.69, 462.61, 148) mm, rotated rx 180 ry 0 rz 160 deg; joints [1.566, 50.675, 8.652, -155.32, 61.678, 167.701]
  Set speed (16.8 mm/s)
  Call Extruder(986.43582)
  MoveL 8331 to (475.11, 461.65, 148) mm, rotated rx 180 ry 0 rz 160 deg; joints [1.432, 50.88, 8.246, -155.423, 61.467, 167.677]
  Set speed (16.8 mm/s)
  Call Extruder(992.04406)
  MoveL 8332 to (476.53, 460.77, 148) mm, rotated rx 180 ry 0 rz 160 deg; joints [1.308, 51.087, 7.838, -155.515, 61.257, 167.648]
  Set speed (16.8 mm/s)
  Call Extruder(997.64409)
  MoveL 8333 to (477.98, 459.94, 148) mm, rotated rx -180 ry 0 rz 160 deg; joints [1.192, 51.3, 7.418, -155.598, 61.044, 167.612]
  Set speed (16.8 mm/s)
  Call Extruder(1003.33329)
  MoveL 8334 to (479.48, 459.14, 148) mm, rotated rx 180 ry 0 rz 160 deg; joints [1.082, 51.522, 6.981, -155.671, 60.824, 167.57]
  Set speed (16.8 mm/s)
  Call Extruder(1008.99762)
  MoveL 8335 to (481, 458.41, 148) mm, rotated rx 180 ry 0 rz 160 deg; joints [0.981, 51.749, 6.534, -155.733, 60.602, 167.522]
  Set speed (16.8 mm/s)
  Call Extruder(1014.56658)
  MoveL 8336 to (482.53, 457.75, 148) mm, rotated rx 180 ry 0 rz 160 deg; joints [0.89, 51.976, 6.084, -155.784, 60.38, 167.468]
  Set speed (16.8 mm/s)
  Call Extruder(1020.29924)
  MoveL 8337 to (484.12, 457.13, 148) mm, rotated rx 180 ry 0 rz 160 deg; joints [0.804, 52.216, 5.612, -155.826, 60.149, 167.406]
  Call Extruder(1025.84043)
  MoveL 8338 to (485.68, 456.58, 148) mm, rotated rx -180 ry 0 rz 160 deg; joints [0.73, 52.453, 5.146, -155.856, 59.924, 167.339]
  Set speed (16.8 mm/s)
  Call Extruder(1031.58175)
  MoveL 8339 to (487.32, 456.08, 148) mm, rotated rx -180 ry 0 rz 160 deg; joints [0.661, 52.702, 4.655, -155.876, 59.688, 167.264]
  Call Extruder(1037.13076)
  MoveL 8340 to (488.91, 455.65, 148) mm, rotated rx 180 ry 0 rz 160 deg; joints [0.602, 52.947, 4.173, -155.886, 59.459, 167.185]
  Set speed (16.8 mm/s)
  Call Extruder(1042.82790)
  MoveL 8341 to (490.57, 455.26, 148) mm, rotated rx 180 ry 0 rz 160 deg; joints [0.55, 53.203, 3.669, -155.885, 59.221, 167.098]
  Set speed (16.8 mm/s)
  Call Extruder(1048.43309)
  MoveL 8342 to (492.21, 454.95, 148) mm, rotated rx -180 ry 0 rz 160 deg; joints [0.507, 53.458, 3.168, -155.873, 58.986, 167.006]
  Set speed (16.8 mm/s)
  Call Extruder(1053.95697)
  MoveL 8343 to (493.84, 454.7, 148) mm, rotated rx -180 ry 0 rz 160 deg; joints [0.473, 53.713, 2.667, -155.852, 58.754, 166.908]
  Set speed (16.8 mm/s)
  Call Extruder(1059.74763)
  MoveL 8344 to (495.56, 454.5, 148) mm, rotated rx -180 ry 0 rz 160 deg; joints [0.445, 53.983, 2.137, -155.818, 58.511, 166.8]
  Set speed (16.8 mm/s)
  Call Extruder(1065.34426)
  MoveL 8345 to (497.22, 454.37, 148) mm, rotated rx -180 ry 0 rz 160 deg; joints [0.426, 54.246, 1.62, -155.776, 58.275, 166.689]
  Set speed (16.8 mm/s)
  Call Extruder(1071.01312)
  MoveL 8346 to (498.91, 454.29, 148) mm, rotated rx -180 ry 0 rz 160 deg; joints [0.416, 54.515, 1.092, -155.722, 58.036, 166.57]
  Set speed (16.8 mm/s)
  Call Extruder(1076.33626)
  MoveL 8347 to (500.5, 454.28, 148) mm, rotated rx 180 ry 0 rz 160 deg; joints [0.413, 54.77, 0.593, -155.662, 57.812, 166.453]
  Set speed (16.8 mm/s)
  Call Extruder(1082.36582)
  MoveL 8348 to (502.3, 454.34, 148) mm, rotated rx -180 ry 0 rz 160 deg; joints [0.418, 55.06, 0.024, -155.583, 57.559, 166.314]
  Set speed (16.8 mm/s)
  Call Extruder(1087.89800)
  MoveL 8349 to (503.95, 454.45, 148) mm, rotated rx 180 ry 0 rz 160 deg; joints [0.431, 55.327, -0.501, -155.5, 57.329, 166.179]
  Set speed (16.8 mm/s)
  Call Extruder(1093.60357)
  MoveL 8350 to (505.64, 454.63, 148) mm, rotated rx 180 ry 0 rz 160 deg; joints [0.452, 55.604, -1.043, -155.405, 57.092, 166.035]
  Call Extruder(1099.21006)
  MoveL 8351 to (507.3, 454.87, 148) mm, rotated rx 180 ry 0 rz 160 deg; joints [0.48, 55.876, -1.577, -155.302, 56.861, 165.887]
  Set speed (16.8 mm/s)
  Call Extruder(1104.88214)
  MoveL 8352 to (508.96, 455.17, 148) mm, rotated rx -180 ry 0 rz 160 deg; joints [0.516, 56.152, -2.117, -155.187, 56.63, 165.732]
  Set speed (16.8 mm/s)
  Call Extruder(1110.20988)
  MoveL 8353 to (510.51, 455.51, 148) mm, rotated rx 180 ry 0 rz 160 deg; joints [0.556, 56.411, -2.624, -155.071, 56.415, 165.581]
  Set speed (16.8 mm/s)
  Call Extruder(1116.11033)
  MoveL 8354 to (512.22, 455.94, 148) mm, rotated rx -180 ry 0 rz 160 deg; joints [0.608, 56.698, -3.185, -154.934, 56.179, 165.408]
  Set speed (16.8 mm/s)
  Call Extruder(1121.81186)
  MoveL 8355 to (513.85, 456.43, 148) mm, rotated rx 180 ry 0 rz 160 deg; joints [0.666, 56.974, -3.725, -154.79, 55.955, 165.235]
  Set speed (16.8 mm/s)
  Call Extruder(1127.46814)
  MoveL 8356 to (515.45, 456.97, 148) mm, rotated rx -180 ry 0 rz 160 deg; joints [0.731, 57.246, -4.258, -154.64, 55.736, 165.058]
  Set speed (16.8 mm/s)
  Call Extruder(1133.03317)
  MoveL 8357 to (517, 457.56, 148) mm, rotated rx 180 ry 0 rz 160 deg; joints [0.8, 57.513, -4.78, -154.483, 55.524, 164.88]
  Set speed (16.8 mm/s)
  Call Extruder(1138.76263)
  MoveL 8358 to (518.57, 458.23, 148) mm, rotated rx -180 ry 0 rz 160 deg; joints [0.879, 57.786, -5.313, -154.313, 55.31, 164.691]
  Call Extruder(1144.32577)
  MoveL 8359 to (520.08, 458.93, 148) mm, rotated rx -180 ry 0 rz 160 deg; joints [0.962, 58.048, -5.826, -154.14, 55.106, 164.503]
  Set speed (16.8 mm/s)
  Call Extruder(1149.95553)
  MoveL 8360 to (521.57, 459.69, 148) mm, rotated rx 180 ry 0 rz 160 deg; joints [1.052, 58.312, -6.34, -153.958, 54.905, 164.308]
  Call Extruder(1155.63325)
  MoveL 8361 to (523.05, 460.52, 148) mm, rotated rx -180 ry 0 rz 160 deg; joints [1.149, 58.574, -6.852, -153.766, 54.707, 164.107]
  Set speed (16.8 mm/s)
  Call Extruder(1161.24123)
  MoveL 8362 to (524.48, 461.39, 148) mm, rotated rx -180 ry 0 rz 160 deg; joints [1.251, 58.83, -7.351, -153.569, 54.517, 163.905]
  Call Extruder(1166.84267)
  MoveL 8363 to (525.88, 462.31, 148) mm, rotated rx 180 ry 0 rz 160 deg; joints [1.358, 59.082, -7.842, -153.366, 54.333, 163.7]
  Call Extruder(1172.53415)
  MoveL 8364 to (527.26, 463.3, 148) mm, rotated rx 180 ry 0 rz 160 deg; joints [1.473, 59.334, -8.334, -153.153, 54.151, 163.488]
  Set speed (16.8 mm/s)
  Call Extruder(1178.25479)
  MoveL 8365 to (528.61, 464.34, 148) mm, rotated rx -180 ry 0 rz 160 deg; joints [1.594, 59.582, -8.818, -152.933, 53.976, 163.272]
  Set speed (16.8 mm/s)
  Call Extruder(1183.79660)
  MoveL 8366 to (529.88, 465.4, 148) mm, rotated rx 180 ry 0 rz 160 deg; joints [1.716, 59.818, -9.278, -152.713, 53.812, 163.061]
  Set speed (16.8 mm/s)
  Call Extruder(1189.48917)
  MoveL 8367 to (531.14, 466.53, 148) mm, rotated rx 180 ry 0 rz 160 deg; joints [1.846, 60.055, -9.74, -152.482, 53.65, 162.84]
  Set speed (16.8 mm/s)
  Call Extruder(1195.09228)
  MoveL 8368 to (532.35, 467.69, 148) mm, rotated rx 180 ry 0 rz 160 deg; joints [1.98, 60.283, -10.185, -152.25, 53.498, 162.622]
  Set speed (16.8 mm/s)
  Call Extruder(1198.06706)
  MoveL 8369 to (532.97, 468.32, 148) mm, rotated rx -180 ry 0 rz 160 deg; joints [2.052, 60.402, -10.416, -152.125, 53.421, 162.505]
  Call Extruder(1201.17613)
  MoveL 8370 to (533.6, 469, 148) mm, rotated rx -180 ry 0 rz 160 deg; joints [2.13, 60.524, -10.654, -151.993, 53.342, 162.383]
  Set speed (16.8 mm/s)
  Call Extruder(1204.28793)
  MoveL 8371 to (534.23, 469.69, 148) mm, rotated rx -180 ry 0 rz 160 deg; joints [2.208, 60.644, -10.888, -151.859, 53.265, 162.26]
  Set speed (16.8 mm/s)
  Call Extruder(1207.45076)
  MoveL 8372 to (534.84, 470.4, 148) mm, rotated rx 180 ry 0 rz 160 deg; joints [2.29, 60.765, -11.123, -151.722, 53.19, 162.135]
  Set speed (16.8 mm/s)
  Call Extruder(1210.56033)
  MoveL 8373 to (535.44, 471.12, 148) mm, rotated rx -180 ry 0 rz 160 deg; joints [2.371, 60.881, -11.349, -151.586, 53.118, 162.011]
  Set speed (16.8 mm/s)
  Call Extruder(1213.69872)
  MoveL 8374 to (536.02, 471.85, 148) mm, rotated rx 180 ry 0 rz 160 deg; joints [2.455, 60.997, -11.574, -151.448, 53.047, 161.887]
  Set speed (16.8 mm/s)
  Call Extruder(1216.97510)
  MoveL 8375 to (536.62, 472.62, 148) mm, rotated rx 180 ry 0 rz 160 deg; joints [2.543, 61.115, -11.804, -151.303, 52.977, 161.757]
  Set speed (16.8 mm/s)
  Call Extruder(1220.00211)
  MoveL 8376 to (537.15, 473.35, 148) mm, rotated rx -180 ry 0 rz 160 deg; joints [2.626, 61.221, -12.011, -151.167, 52.915, 161.636]
  Call Extruder(1223.07974)
  MoveL 8377 to (537.68, 474.1, 148) mm, rotated rx 180 ry 0 rz 160 deg; joints [2.711, 61.328, -12.218, -151.029, 52.853, 161.514]
  Set speed (16.8 mm/s)
  Call Extruder(1226.23291)
  MoveL 8378 to (538.2, 474.88, 148) mm, rotated rx 180 ry 0 rz 160 deg; joints [2.8, 61.434, -12.426, -150.886, 52.794, 161.389]
  Set speed (16.8 mm/s)
  Call Extruder(1229.52531)
  MoveL 8379 to (538.73, 475.71, 148) mm, rotated rx 180 ry 0 rz 160 deg; joints [2.893, 61.544, -12.638, -150.737, 52.734, 161.258]
  Call Extruder(1232.52102)
  MoveL 8380 to (539.2, 476.47, 148) mm, rotated rx 180 ry 0 rz 160 deg; joints [2.98, 61.64, -12.825, -150.6, 52.682, 161.14]
  Set speed (16.8 mm/s)
  Call Extruder(1235.63407)
  MoveL 8381 to (539.67, 477.27, 148) mm, rotated rx -180 ry 0 rz 160 deg; joints [3.07, 61.738, -13.016, -150.457, 52.631, 161.017]
  Set speed (16.8 mm/s)
  Call Extruder(1240.93493)
  MoveL 8382 to (540.43, 478.65, 148) mm, rotated rx -180 ry 0 rz 160 deg; joints [3.227, 61.899, -13.329, -150.214, 52.55, 160.809]
  Set speed (16.8 mm/s)
  Call Extruder(1245.07482)
  MoveL 8383 to (540.99, 479.75, 148) mm, rotated rx -180 ry 0 rz 160 deg; joints [3.351, 62.019, -13.563, -150.022, 52.493, 160.648]
  Set speed (16.8 mm/s)
  Call Extruder(1248.20774)
  MoveL 8384 to (541.4, 480.6, 148) mm, rotated rx -180 ry 0 rz 160 deg; joints [3.447, 62.107, -13.733, -149.877, 52.452, 160.527]
  Set speed (16.8 mm/s)
  Call Extruder(1251.52933)
  MoveL 8385 to (541.81, 481.5, 148) mm, rotated rx -180 ry 0 rz 160 deg; joints [3.549, 62.198, -13.909, -149.723, 52.413, 160.399]
  Call Extruder(1257.63197)
  MoveL 8386 to (542.51, 483.18, 148) mm, rotated rx -180 ry 0 rz 160 deg; joints [3.738, 62.355, -14.215, -149.439, 52.349, 160.166]
  Set speed (16.8 mm/s)
  Call Extruder(1263.78798)
  MoveL 8387 to (543.15, 484.9, 148) mm, rotated rx -180 ry 0 rz 160 deg; joints [3.933, 62.503, -14.502, -149.153, 52.295, 159.935]
  Set speed (16.8 mm/s)
  Call Extruder(1267.17533)
  MoveL 8388 to (543.47, 485.86, 148) mm, rotated rx 180 ry 0 rz 160 deg; joints [4.041, 62.579, -14.65, -148.997, 52.271, 159.81]
  Call Extruder(1270.15440)
  MoveL 8389 to (543.74, 486.7, 148) mm, rotated rx -180 ry 0 rz 160 deg; joints [4.137, 62.644, -14.776, -148.859, 52.252, 159.701]
  Call Extruder(1273.43411)
  MoveL 8390 to (544.01, 487.64, 148) mm, rotated rx -180 ry 0 rz 160 deg; joints [4.243, 62.71, -14.905, -148.708, 52.235, 159.582]
  Call Extruder(1276.57248)
  MoveL 8391 to (544.26, 488.54, 148) mm, rotated rx 180 ry 0 rz 160 deg; joints [4.345, 62.772, -15.026, -148.563, 52.221, 159.47]
  Set speed (16.8 mm/s)
  Call Extruder(1282.88416)
  MoveL 8392 to (544.7, 490.37, 148) mm, rotated rx -180 ry 0 rz 160 deg; joints [4.552, 62.886, -15.247, -148.274, 52.202, 159.248]
  Set speed (16.8 mm/s)
  Call Extruder(1289.17171)
  MoveL 8393 to (545.05, 492.22, 148) mm, rotated rx -180 ry 0 rz 160 deg; joints [4.761, 62.987, -15.442, -147.988, 52.197, 159.034]
  Set speed (16.8 mm/s)
  Call Extruder(1295.42805)
  MoveL 8394 to (545.33, 494.06, 148) mm, rotated rx 180 ry 0 rz 160 deg; joints [4.971, 63.074, -15.611, -147.707, 52.203, 158.827]
  Set speed (16.8 mm/s)
  Call Extruder(1301.72546)
  MoveL 8395 to (545.54, 495.93, 148) mm, rotated rx 180 ry 0 rz 160 deg; joints [5.183, 63.148, -15.755, -147.428, 52.221, 158.626]
  Set speed (16.8 mm/s)
  Call Extruder(1307.96140)
  MoveL 8396 to (545.67, 497.78, 148) mm, rotated rx -180 ry 0 rz 160 deg; joints [5.395, 63.207, -15.87, -147.155, 52.251, 158.435]
  Call Extruder(1314.23549)
  MoveL 8397 to (545.72, 499.66, 148) mm, rotated rx 180 ry 0 rz 160 deg; joints [5.609, 63.254, -15.96, -146.885, 52.294, 158.251]
  Set speed (16.8 mm/s)
  Call Extruder(1320.59919)
  MoveL 8398 to (545.69, 501.55, 148) mm, rotated rx -180 ry 0 rz 160 deg; joints [5.827, 63.287, -16.024, -146.616, 52.349, 158.073]
  Set speed (16.8 mm/s)
  Call Extruder(1326.76905)
  MoveL 8399 to (545.59, 503.39, 148) mm, rotated rx 180 ry 0 rz 160 deg; joints [6.039, 63.305, -16.06, -146.361, 52.414, 157.91]
  Call Extruder(1332.78282)
  MoveL 8400 to (545.42, 505.18, 148) mm, rotated rx -180 ry 0 rz 160 deg; joints [6.245, 63.31, -16.068, -146.118, 52.488, 157.76]
  Set speed (16.8 mm/s)
  Call Extruder(1339.39723)
  MoveL 8401 to (545.16, 507.14, 148) mm, rotated rx -180 ry 0 rz 160 deg; joints [6.473, 63.3, -16.051, -145.857, 52.582, 157.605]
  Set speed (16.8 mm/s)
  Call Extruder(1345.55974)
  MoveL 8402 to (544.83, 508.95, 148) mm, rotated rx 180 ry 0 rz 160 deg; joints [6.684, 63.277, -16.005, -145.62, 52.681, 157.471]
  Call Extruder(1351.83207)
  MoveL 8403 to (544.43, 510.78, 148) mm, rotated rx 180 ry 0 rz 160 deg; joints [6.898, 63.24, -15.934, -145.386, 52.792, 157.345]
  Set speed (16.8 mm/s)
  Call Extruder(1354.92811)
  MoveL 8404 to (544.2, 511.67, 148) mm, rotated rx -180 ry 0 rz 160 deg; joints [7.004, 63.216, -15.887, -145.274, 52.851, 157.288]
  Set speed (16.8 mm/s)
  Call Extruder(1358.91243)
  MoveL 8405 to (543.89, 512.81, 148) mm, rotated rx -180 ry 0 rz 160 deg; joints [7.139, 63.183, -15.823, -145.131, 52.929, 157.216]
  Set speed (16.8 mm/s)
  Call Extruder(1364.33583)
  MoveL 8406 to (543.41, 514.36, 148) mm, rotated rx -180 ry 0 rz 160 deg; joints [7.323, 63.126, -15.711, -144.943, 53.044, 157.127]
  Set speed (16.8 mm/s)
  Call Extruder(1370.52426)
  MoveL 8407 to (542.79, 516.1, 148) mm, rotated rx 180 ry 0 rz 160 deg; joints [7.531, 63.049, -15.562, -144.734, 53.184, 157.035]
  Set speed (16.8 mm/s)
  Call Extruder(1376.67051)
  MoveL 8408 to (542.11, 517.8, 148) mm, rotated rx 180 ry 0 rz 160 deg; joints [7.736, 62.96, -15.39, -144.534, 53.333, 156.954]
  Set speed (16.8 mm/s)
  Call Extruder(1383.03982)
  MoveL 8409 to (541.34, 519.53, 148) mm, rotated rx 180 ry 0 rz 160 deg; joints [7.947, 62.854, -15.184, -144.336, 53.497, 156.883]
  Set speed (16.8 mm/s)
  Call Extruder(1386.11259)
  MoveL 8410 to (540.94, 520.36, 148) mm, rotated rx 180 ry 0 rz 160 deg; joints [8.048, 62.798, -15.076, -144.243, 53.579, 156.852]
  Set speed (16.8 mm/s)
  Call Extruder(1389.83367)
  MoveL 8411 to (540.43, 521.35, 148) mm, rotated rx 180 ry 0 rz 160 deg; joints [8.17, 62.727, -14.937, -144.133, 53.681, 156.819]
  Call Extruder(1395.48705)
  MoveL 8412 to (539.62, 522.82, 148) mm, rotated rx 180 ry 0 rz 160 deg; joints [8.353, 62.61, -14.71, -143.972, 53.843, 156.776]
  Set speed (16.8 mm/s)
  Call Extruder(1398.79433)
  MoveL 8413 to (539.12, 523.68, 148) mm, rotated rx -180 ry 0 rz 160 deg; joints [8.459, 62.537, -14.568, -143.881, 53.94, 156.754]
  Set speed (16.8 mm/s)
  Call Extruder(1402.61611)
  MoveL 8414 to (538.51, 524.64, 148) mm, rotated rx 180 ry 0 rz 160 deg; joints [8.58, 62.447, -14.395, -143.779, 54.056, 156.735]
  Set speed (16.8 mm/s)
  Call Extruder(1405.06550)
  MoveL 8415 to (538.11, 525.25, 148) mm, rotated rx 180 ry 0 rz 160 deg; joints [8.657, 62.388, -14.279, -143.715, 54.132, 156.724]
  Call Extruder(1408.06249)
  MoveL 8416 to (537.61, 526, 148) mm, rotated rx -180 ry 0 rz 160 deg; joints [8.751, 62.314, -14.134, -143.639, 54.225, 156.714]
  Set speed (16.8 mm/s)
  Call Extruder(1411.99980)
  MoveL 8417 to (536.93, 526.95, 148) mm, rotated rx 180 ry 0 rz 160 deg; joints [8.874, 62.211, -13.936, -143.542, 54.351, 156.703]
  Set speed (16.8 mm/s)
  Call Extruder(1417.45738)
  MoveL 8418 to (535.95, 528.25, 148) mm, rotated rx 180 ry 0 rz 160 deg; joints [9.041, 62.062, -13.645, -143.413, 54.531, 156.697]
  Set speed (16.8 mm/s)
  Call Extruder(1420.74924)
  MoveL 8419 to (535.33, 529.02, 148) mm, rotated rx -180 ry 0 rz 160 deg; joints [9.141, 61.968, -13.463, -143.338, 54.641, 156.696]
  Set speed (16.8 mm/s)
  Call Extruder(1423.89732)
  MoveL 8420 to (534.73, 529.74, 148) mm, rotated rx -180 ry 0 rz 160 deg; joints [9.235, 61.875, -13.283, -143.269, 54.749, 156.699]
  Set speed (16.8 mm/s)
  Call Extruder(1426.87652)
  MoveL 8421 to (534.14, 530.4, 148) mm, rotated rx 180 ry 0 rz 160 deg; joints [9.323, 61.785, -13.107, -143.206, 54.852, 156.705]
  Set speed (16.8 mm/s)
  Call Extruder(1430.17860)
  MoveL 8422 to (533.48, 531.13, 148) mm, rotated rx -180 ry 0 rz 160 deg; joints [9.42, 61.682, -12.907, -143.138, 54.968, 156.713]
  Call Extruder(1433.17911)
  MoveL 8423 to (532.87, 531.78, 148) mm, rotated rx -180 ry 0 rz 160 deg; joints [9.507, 61.586, -12.721, -143.079, 55.075, 156.724]
  Set speed (16.8 mm/s)
  Call Extruder(1436.28830)
  MoveL 8424 to (532.21, 532.44, 148) mm, rotated rx 180 ry 0 rz 160 deg; joints [9.595, 61.484, -12.523, -143.02, 55.187, 156.737]
  Call Extruder(1439.42622)
  MoveL 8425 to (531.54, 533.09, 148) mm, rotated rx 180 ry 0 rz 160 deg; joints [9.684, 61.379, -12.318, -142.962, 55.301, 156.754]
  Set speed (16.8 mm/s)
  Call Extruder(1442.69654)
  MoveL 8426 to (530.83, 533.76, 148) mm, rotated rx 180 ry 0 rz 160 deg; joints [9.775, 61.268, -12.101, -142.904, 55.421, 156.773]
  Set speed (16.8 mm/s)
  Call Extruder(1445.72772)
  MoveL 8427 to (530.16, 534.36, 148) mm, rotated rx -180 ry 0 rz 160 deg; joints [9.859, 61.161, -11.894, -142.853, 55.534, 156.794]
  Set speed (16.8 mm/s)
  Call Extruder(1448.79219)
  MoveL 8428 to (529.46, 534.96, 148) mm, rotated rx 180 ry 0 rz 160 deg; joints [9.942, 61.052, -11.681, -142.803, 55.65, 156.817]
  Set speed (16.8 mm/s)
  Call Extruder(1453.72387)
  MoveL 8429 to (528.32, 535.89, 148) mm, rotated rx -180 ry 0 rz 160 deg; joints [10.074, 60.872, -11.331, -142.727, 55.837, 156.86]
  Set speed (16.9 mm/s)
  Call Extruder(1458.95401)
  MoveL 8430 to (527.08, 536.84, 148) mm, rotated rx 180 ry 0 rz 160 deg; joints [10.21, 60.674, -10.946, -142.652, 56.039, 156.912]
  Set speed (16.8 mm/s)
  Call Extruder(1464.46698)
  MoveL 8431 to (525.74, 537.79, 148) mm, rotated rx -180 ry 0 rz 160 deg; joints [10.349, 60.46, -10.529, -142.581, 56.255, 156.974]
  Set speed (16.8 mm/s)
  Call Extruder(1467.80952)
  MoveL 8432 to (524.91, 538.34, 148) mm, rotated rx 180 ry 0 rz 160 deg; joints [10.431, 60.328, -10.271, -142.541, 56.387, 157.015]
  Set speed (16.8 mm/s)
  Call Extruder(1470.74806)
  MoveL 8433 to (524.17, 538.81, 148) mm, rotated rx -180 ry 0 rz 160 deg; joints [10.502, 60.209, -10.041, -142.507, 56.503, 157.054]
  Set speed (16.8 mm/s)
  Call Extruder(1474.00772)
  MoveL 8434 to (523.34, 539.32, 148) mm, rotated rx -180 ry 0 rz 160 deg; joints [10.58, 60.076, -9.782, -142.473, 56.633, 157.099]
  Set speed (16.8 mm/s)
  Call Extruder(1479.66394)
  MoveL 8435 to (521.87, 540.15, 148) mm, rotated rx -180 ry 0 rz 160 deg; joints [10.71, 59.841, -9.324, -142.419, 56.861, 157.183]
  Set speed (16.8 mm/s)
  Call Extruder(1483.26855)
  MoveL 8436 to (520.92, 540.65, 148) mm, rotated rx 180 ry 0 rz 160 deg; joints [10.79, 59.689, -9.026, -142.388, 57.007, 157.24]
  Call Extruder(1486.57376)
  MoveL 8437 to (520.04, 541.09, 148) mm, rotated rx -180 ry 0 rz 160 deg; joints [10.861, 59.547, -8.75, -142.362, 57.141, 157.295]
  Call Extruder(1489.76395)
  MoveL 8438 to (519.18, 541.5, 148) mm, rotated rx -180 ry 0 rz 160 deg; joints [10.929, 59.409, -8.481, -142.339, 57.271, 157.35]
  Set speed (16.8 mm/s)
  Call Extruder(1496.07580)
  MoveL 8439 to (517.46, 542.26, 148) mm, rotated rx 180 ry 0 rz 160 deg; joints [11.058, 59.131, -7.939, -142.302, 57.529, 157.466]
  Set speed (16.8 mm/s)
  Call Extruder(1501.98790)
  MoveL 8440 to (515.81, 542.9, 148) mm, rotated rx -180 ry 0 rz 160 deg; joints [11.172, 58.865, -7.42, -142.275, 57.773, 157.582]
  Set speed (16.8 mm/s)
  Call Extruder(1504.60189)
  MoveL 8441 to (515.08, 543.16, 148) mm, rotated rx -180 ry 0 rz 160 deg; joints [11.22, 58.747, -7.19, -142.265, 57.88, 157.635]
  Set speed (16.8 mm/s)
  Call Extruder(1508.35148)
  MoveL 8442 to (514.02, 543.52, 148) mm, rotated rx 180 ry 0 rz 160 deg; joints [11.288, 58.576, -6.856, -142.254, 58.034, 157.713]
  Set speed (16.8 mm/s)
  Call Extruder(1514.07736)
  MoveL 8443 to (512.39, 544.02, 148) mm, rotated rx -180 ry 0 rz 160 deg; joints [11.386, 58.312, -6.341, -142.242, 58.27, 157.838]
  Set speed (16.8 mm/s)
  Call Extruder(1520.84517)
  MoveL 8444 to (510.43, 544.51, 148) mm, rotated rx 180 ry 0 rz 160 deg; joints [11.493, 57.995, -5.721, -142.24, 58.549, 157.995]
  Call Extruder(1527.39442)
  MoveL 8445 to (508.52, 544.92, 148) mm, rotated rx 180 ry 0 rz 160 deg; joints [11.588, 57.685, -5.116, -142.247, 58.819, 158.153]
  Set speed (16.8 mm/s)
  Call Extruder(1533.74644)
  MoveL 8446 to (506.65, 545.23, 148) mm, rotated rx 180 ry 0 rz 160 deg; joints [11.672, 57.382, -4.524, -142.262, 59.079, 158.312]
  Call Extruder(1539.67102)
  MoveL 8447 to (504.9, 545.46, 148) mm, rotated rx -180 ry 0 rz 160 deg; joints [11.743, 57.097, -3.967, -142.285, 59.32, 158.467]
  Set speed (16.8 mm/s)
  Call Extruder(1546.23868)
  MoveL 8448 to (502.95, 545.62, 148) mm, rotated rx -180 ry 0 rz 160 deg; joints [11.813, 56.78, -3.346, -142.319, 59.585, 158.644]
  Set speed (16.8 mm/s)
  Call Extruder(1552.53415)
  MoveL 8449 to (501.07, 545.71, 148) mm, rotated rx -180 ry 0 rz 160 deg; joints [11.871, 56.475, -2.749, -142.361, 59.838, 158.819]
  Set speed (16.8 mm/s)
  Call Extruder(1558.74230)
  MoveL 8450 to (499.22, 545.71, 148) mm, rotated rx 180 ry 0 rz 160 deg; joints [11.919, 56.173, -2.158, -142.411, 60.084, 158.997]
  Set speed (10.0 mm/s)
  MoveL 8451 to (499.22, 545.71, 152) mm, rotated rx 180 ry 0 rz 160 deg; joints [11.919, 55.599, -2.014, -142.258, 59.744, 158.693]
  Set speed (120.0 mm/s)
  MoveL 8452 to (499.29, 544.23, 152) mm, rotated rx -180 ry 0 rz 160 deg; joints [11.736, 55.559, -1.936, -142.47, 59.707, 158.82]
  Set speed (16.9 mm/s)
  Call Extruder(1564.83219)
  MoveL 8453 to (497.46, 544.16, 152) mm, rotated rx 180 ry 0 rz 160 deg; joints [11.774, 55.26, -1.354, -142.529, 59.946, 158.999]
  Set speed (16.9 mm/s)
  Call Extruder(1570.91488)
  MoveL 8454 to (495.65, 544.02, 152) mm, rotated rx 180 ry 0 rz 160 deg; joints [11.803, 54.961, -0.773, -142.596, 60.18, 159.181]
  Call Extruder(0.00000)
  Call Extruder(5.96228)
  MoveL 8455 to (493.87, 543.81, 152) mm, rotated rx -180 ry 0 rz 160 deg; joints [11.823, 54.669, -0.204, -142.671, 60.407, 159.364]
  Set speed (16.9 mm/s)
  Call Extruder(11.95792)
  MoveL 8456 to (492.1, 543.52, 152) mm, rotated rx 180 ry 0 rz 160 deg; joints [11.834, 54.377, 0.366, -142.754, 60.632, 159.551]
  Call Extruder(17.78507)
  MoveL 8457 to (490.39, 543.17, 152) mm, rotated rx 180 ry 0 rz 160 deg; joints [11.835, 54.094, 0.917, -142.844, 60.846, 159.736]
  Set speed (16.9 mm/s)
  Call Extruder(21.08852)
  MoveL 8458 to (489.42, 542.95, 152) mm, rotated rx 180 ry 0 rz 160 deg; joints [11.832, 53.935, 1.228, -142.898, 60.965, 159.842]
  Call Extruder(23.81430)
  MoveL 8459 to (488.63, 542.75, 152) mm, rotated rx -180 ry 0 rz 160 deg; joints [11.828, 53.804, 1.483, -142.944, 61.063, 159.93]
  Set speed (16.9 mm/s)
  Call Extruder(29.88548)
  MoveL 8460 to (486.88, 542.24, 152) mm, rotated rx 180 ry 0 rz 160 deg; joints [11.81, 53.513, 2.048, -143.054, 61.277, 160.129]
  Call Extruder(35.91080)
  MoveL 8461 to (485.17, 541.67, 152) mm, rotated rx -180 ry 0 rz 160 deg; joints [11.783, 53.228, 2.604, -143.171, 61.485, 160.327]
  Call Extruder(42.09194)
  MoveL 8462 to (483.44, 541.02, 152) mm, rotated rx 180 ry 0 rz 160 deg; joints [11.746, 52.939, 3.168, -143.3, 61.692, 160.534]
  Set speed (16.9 mm/s)
  Call Extruder(46.74493)
  MoveL 8463 to (482.15, 540.48, 152) mm, rotated rx 180 ry 0 rz 160 deg; joints [11.711, 52.725, 3.587, -143.403, 61.845, 160.69]
  Set speed (16.9 mm/s)
  Call Extruder(51.12671)
  MoveL 8464 to (480.96, 539.93, 152) mm, rotated rx -180 ry 0 rz 160 deg; joints [11.672, 52.525, 3.977, -143.505, 61.985, 160.837]
  Set speed (16.9 mm/s)
  Call Extruder(55.68037)
  MoveL 8465 to (479.74, 539.32, 152) mm, rotated rx 180 ry 0 rz 160 deg; joints [11.628, 52.319, 4.378, -143.614, 62.127, 160.991]
  Set speed (16.9 mm/s)
  Call Extruder(60.24798)
  MoveL 8466 to (478.53, 538.68, 152) mm, rotated rx 180 ry 0 rz 160 deg; joints [11.576, 52.116, 4.775, -143.73, 62.267, 161.147]
  Set speed (16.9 mm/s)
  Call Extruder(63.25317)
  MoveL 8467 to (477.75, 538.23, 152) mm, rotated rx 180 ry 0 rz 160 deg; joints [11.54, 51.984, 5.033, -143.808, 62.356, 161.249]
  Set speed (16.9 mm/s)
  Call Extruder(66.20513)
  MoveL 8468 to (476.99, 537.78, 152) mm, rotated rx -180 ry 0 rz 160 deg; joints [11.501, 51.855, 5.285, -143.887, 62.443, 161.35]
  Set speed (16.9 mm/s)
  Call Extruder(69.26499)
  MoveL 8469 to (476.21, 537.29, 152) mm, rotated rx 180 ry 0 rz 160 deg; joints [11.459, 51.723, 5.543, -143.971, 62.532, 161.454]
  Set speed (16.9 mm/s)
  Call Extruder(72.32220)
  MoveL 8470 to (475.44, 536.79, 152) mm, rotated rx 180 ry 0 rz 160 deg; joints [11.414, 51.593, 5.798, -144.057, 62.618, 161.559]
  Set speed (16.9 mm/s)
  Call Extruder(75.32921)
  MoveL 8471 to (474.7, 536.28, 152) mm, rotated rx 180 ry 0 rz 160 deg; joints [11.368, 51.466, 6.045, -144.143, 62.701, 161.661]
  Call Extruder(78.30963)
  MoveL 8472 to (473.97, 535.76, 152) mm, rotated rx 180 ry 0 rz 160 deg; joints [11.319, 51.342, 6.288, -144.231, 62.782, 161.763]
  Set speed (16.9 mm/s)
  Call Extruder(81.47187)
  MoveL 8473 to (473.21, 535.2, 152) mm, rotated rx 180 ry 0 rz 160 deg; joints [11.265, 51.212, 6.543, -144.325, 62.867, 161.871]
  Set speed (16.9 mm/s)
  Call Extruder(84.46560)
  MoveL 8474 to (472.5, 534.65, 152) mm, rotated rx 180 ry 0 rz 160 deg; joints [11.211, 51.09, 6.78, -144.417, 62.944, 161.973]
  Set speed (16.9 mm/s)
  Call Extruder(87.31057)
  MoveL 8475 to (471.84, 534.11, 152) mm, rotated rx 180 ry 0 rz 160 deg; joints [11.159, 50.976, 7.004, -144.506, 63.017, 162.07]
  Set speed (16.9 mm/s)
  Call Extruder(90.44252)
  MoveL 8476 to (471.12, 533.51, 152) mm, rotated rx 180 ry 0 rz 160 deg; joints [11.098, 50.852, 7.246, -144.606, 63.094, 162.176]
  Set speed (16.9 mm/s)
  Call Extruder(93.39837)
  MoveL 8477 to (470.46, 532.92, 152) mm, rotated rx 180 ry 0 rz 160 deg; joints [11.038, 50.737, 7.471, -144.702, 63.166, 162.277]
  Set speed (16.9 mm/s)
  Call Extruder(98.17683)
  MoveL 8478 to (469.41, 531.95, 152) mm, rotated rx 180 ry 0 rz 160 deg; joints [10.937, 50.554, 7.829, -144.861, 63.278, 162.438]
  Call Extruder(102.48403)
  MoveL 8479 to (468.49, 531.04, 152) mm, rotated rx 180 ry 0 rz 160 deg; joints [10.841, 50.394, 8.142, -145.008, 63.375, 162.583]
  Set speed (16.9 mm/s)
  Call Extruder(105.52077)
  MoveL 8480 to (467.86, 530.39, 152) mm, rotated rx -180 ry 0 rz 160 deg; joints [10.77, 50.283, 8.359, -145.114, 63.441, 162.685]
  Set speed (16.9 mm/s)
  Call Extruder(108.59106)
